LIN {X 0,Y 360.428,Z 320.263,A -85,B 0,C 180,E1 -13052.235,E2 -13052.235} C_VEL
LIN {X 0,Y 360.36,Z 319.532,A -85,B 0,C 180,E1 -13053.354,E2 -13053.354} C_VEL
LIN {X 0,Y 360.368,Z 318.39,A -85,B 0,C 180,E1 -13054.474,E2 -13054.474} C_VEL
LIN {X 0,Y 360.408,Z 314.81,A -85,B 0,C 180,E1 -13056.719,E2 -13056.719} C_VEL
LIN {X 0,Y 360.696,Z 310.966,A -85,B 0,C 180,E1 -13058.403,E2 -13058.403} C_VEL
LIN {X 0,Y 361.141,Z 306.012,A -85,B 0,C 180,E1 -13060.087,E2 -13060.087} C_VEL
LIN {X 0,Y 361.815,Z 299.808,A -85,B 0,C 180,E1 -13061.768,E2 -13061.768} C_VEL
LIN {X 0,Y 362.921,Z 292.123,A -85,B 0,C 180,E1 -13063.437,E2 -13063.437} C_VEL
LIN {X 0,Y 363.918,Z 283.845,A -85,B 0,C 180,E1 -13064.897,E2 -13064.897} C_VEL
LIN {X 0,Y 365.211,Z 273.678,A -85,B 0,C 180,E1 -13066.346,E2 -13066.346} C_VEL
LIN {X 0,Y 366.644,Z 262.906,A -85,B 0,C 180,E1 -13067.572,E2 -13067.572} C_VEL
LIN {X 0,Y 367.851,Z 252.444,A -85,B 0,C 180,E1 -13068.52,E2 -13068.52} C_VEL
LIN {X 0,Y 369.117,Z 239.88,A -85,B 0,C 180,E1 -13069.391,E2 -13069.391} C_VEL
LIN {X 0,Y 370.219,Z 226.622,A -85,B 0,C 180,E1 -13070.053,E2 -13070.053} C_VEL
LIN {X 0,Y 370.793,Z 214.493,A -85,B 0,C 180,E1 -13070.455,E2 -13070.455} C_VEL
LIN {X 0,Y 372.141,Z 144.791,A -85,B 0,C 180,E1 -13071.833,E2 -13071.833} C_VEL
LIN {X 0,Y 368.386,Z 121.336,A -85,B 0,C 180,E1 -13072.599,E2 -13072.599} C_VEL
LIN {X 0,Y 365.441,Z 106.485,A -85,B 0,C 180,E1 -13073.16,E2 -13073.16} C_VEL
LIN {X 0,Y 367.084,Z 91.512,A -85,B 0,C 180,E1 -13076.432,E2 -13076.432} C_VEL
LIN {X 0,Y 365.836,Z 84.095,A -85,B 0,C 180,E1 -13078.246,E2 -13078.246} C_VEL
LIN {X 0,Y 363.068,Z 72.33,A -85,B 0,C 180,E1 -13081.298,E2 -13081.298} C_VEL
LIN {X 0,Y 361.872,Z 67.409,A -85,B 0,C 180,E1 -13082.653,E2 -13082.653} C_VEL
LIN {X 0,Y 361.87,Z 67.409,A -85,B 0,C 180,E1 -13085.637,E2 -13085.637} C_VEL
LIN {X 0,Y 361.871,Z 67.398,A -85,B 0,C 180,E1 -13089.027,E2 -13089.027} C_VEL
LIN {X 0,Y 361.839,Z 67.408,A -85,B 0,C 180,E1 -13092.829,E2 -13092.829} C_VEL
LIN {X 0,Y 361.821,Z 67.412,A -85,B 0,C 180,E1 -13095.946,E2 -13095.946} C_VEL
LIN {X 0,Y 361.838,Z 67.41,A -85,B 0,C 180,E1 -13099.245,E2 -13099.245} C_VEL
LIN {X 0,Y 361.866,Z 67.404,A -85,B 0,C 180,E1 -13102.777,E2 -13102.777} C_VEL
LIN {X 0,Y 361.857,Z 67.405,A -85,B 0,C 180,E1 -13105.72,E2 -13105.72} C_VEL
LIN {X 0,Y 361.878,Z 67.401,A -85,B 0,C 180,E1 -13109.672,E2 -13109.672} C_VEL
LIN {X 0,Y 361.958,Z 67.392,A -85,B 0,C 180,E1 -13113.475,E2 -13113.475} C_VEL
LIN {X 0,Y 361.894,Z 67.402,A -85,B 0,C 180,E1 -13117.145,E2 -13117.145} C_VEL
LIN {X 0,Y 361.91,Z 67.405,A -85,B 0,C 180,E1 -13120.723,E2 -13120.723} C_VEL
LIN {X 0,Y 361.936,Z 67.392,A -85,B 0,C 180,E1 -13123.066,E2 -13123.066} C_VEL
LIN {X 0,Y 362.002,Z 67.389,A -85,B 0,C 180,E1 -13126.528,E2 -13126.528} C_VEL
LIN {X 0,Y 362.035,Z 67.387,A -85,B 0,C 180,E1 -13129.938,E2 -13129.938} C_VEL
LIN {X 0,Y 362.165,Z 67.36,A -85,B 0,C 180,E1 -13133.314,E2 -13133.314} C_VEL
LIN {X 0,Y 362.282,Z 67.351,A -85,B 0,C 180,E1 -13137.776,E2 -13137.776} C_VEL
LIN {X 0,Y 362.43,Z 67.338,A -85,B 0,C 180,E1 -13140,E2 -13140} C_VEL
LIN {X 0,Y 362.283,Z 67.353,A -85,B 0,C 180,E1 -13142.223,E2 -13142.223} C_VEL
LIN {X 0,Y 362.15,Z 67.372,A -85,B 0,C 180,E1 -13146.686,E2 -13146.686} C_VEL
LIN {X 0,Y 362.003,Z 67.389,A -85,B 0,C 180,E1 -13150.063,E2 -13150.063} C_VEL
LIN {X 0,Y 362.001,Z 67.383,A -85,B 0,C 180,E1 -13153.899,E2 -13153.899} C_VEL
LIN {X 0,Y 361.931,Z 67.404,A -85,B 0,C 180,E1 -13156.934,E2 -13156.934} C_VEL
LIN {X 0,Y 361.896,Z 67.404,A -85,B 0,C 180,E1 -13160.46,E2 -13160.46} C_VEL
LIN {X 0,Y 361.895,Z 67.401,A -85,B 0,C 180,E1 -13164.113,E2 -13164.113} C_VEL
LIN {X 0,Y 361.867,Z 67.405,A -85,B 0,C 180,E1 -13167.782,E2 -13167.782} C_VEL
LIN {X 0,Y 361.848,Z 67.409,A -85,B 0,C 180,E1 -13171.285,E2 -13171.285} C_VEL
LIN {X 0,Y 361.856,Z 67.408,A -85,B 0,C 180,E1 -13174.28,E2 -13174.28} C_VEL
LIN {X 0,Y 361.862,Z 67.407,A -85,B 0,C 180,E1 -13177.222,E2 -13177.222} C_VEL
LIN {X 0,Y 361.83,Z 67.4,A -85,B 0,C 180,E1 -13180.754,E2 -13180.754} C_VEL
LIN {X 0,Y 361.818,Z 67.416,A -85,B 0,C 180,E1 -13184.368,E2 -13184.368} C_VEL
LIN {X 0,Y 361.836,Z 67.416,A -85,B 0,C 180,E1 -13187.568,E2 -13187.568} C_VEL
LIN {X 0,Y 361.831,Z 67.413,A -85,B 0,C 180,E1 -13190.981,E2 -13190.981} C_VEL
LIN {X 0,Y 361.875,Z 67.411,A -85,B 0,C 180,E1 -13194.655,E2 -13194.655} C_VEL
LIN {X 0,Y 361.926,Z 67.537,A -85,B 0,C 180,E1 -13195.305,E2 -13195.305} C_VEL
LIN {X 0,Y 362.975,Z 72.103,A -85,B 0,C 180,E1 -13196.708,E2 -13196.708} C_VEL
LIN {X 0,Y 372.386,Z 94.109,A -85,B 0,C 180,E1 -13197.911,E2 -13197.911} C_VEL
LIN {X 0,Y 373.147,Z 96.414,A -85,B 0,C 180,E1 -13198.016,E2 -13198.016} C_VEL
LIN {X 0,Y 371.369,Z 178.271,A -85,B 0,C 180,E1 -13199.626,E2 -13199.626} C_VEL
LIN {X 0,Y 370.873,Z 191.183,A -85,B 0,C 180,E1 -13200.091,E2 -13200.091} C_VEL
LIN {X 0,Y 370.25,Z 203.565,A -85,B 0,C 180,E1 -13200.76,E2 -13200.76} C_VEL
LIN {X 0,Y 369.334,Z 215.148,A -85,B 0,C 180,E1 -13201.594,E2 -13201.594} C_VEL
LIN {X 0,Y 368.036,Z 227.162,A -85,B 0,C 180,E1 -13202.722,E2 -13202.722} C_VEL
LIN {X 0,Y 366.749,Z 238.059,A -85,B 0,C 180,E1 -13204.027,E2 -13204.027} C_VEL
LIN {X 0,Y 365.655,Z 246.559,A -85,B 0,C 180,E1 -13205.289,E2 -13205.289} C_VEL
LIN {X 0,Y 364.569,Z 254.494,A -85,B 0,C 180,E1 -13206.722,E2 -13206.722} C_VEL
LIN {X 0,Y 363.432,Z 262.175,A -85,B 0,C 180,E1 -13208.443,E2 -13208.443} C_VEL
LIN {X 0,Y 362.508,Z 268.298,A -85,B 0,C 180,E1 -13210.167,E2 -13210.167} C_VEL
LIN {X 0,Y 361.747,Z 273.775,A -85,B 0,C 180,E1 -13212.17,E2 -13212.17} C_VEL
LIN {X 0,Y 361.11,Z 277.706,A -85,B 0,C 180,E1 -13214.189,E2 -13214.189} C_VEL
LIN {X 0,Y 360.871,Z 279.318,A -85,B 0,C 180,E1 -13215.334,E2 -13215.334} C_VEL
LIN {X 0,Y 360.663,Z 280.878,A -85,B 0,C 180,E1 -13216.986,E2 -13216.986} C_VEL
LIN {X 0,Y 360.463,Z 281.603,A -85,B 0,C 180,E1 -13218.757,E2 -13218.757} C_VEL
LIN {X 0,Y 360.418,Z 281.121,A -85,B 0,C 180,E1 -13221.025,E2 -13221.025} C_VEL
LIN {X 0,Y 360.479,Z 280.243,A -85,B 0,C 180,E1 -13222.156,E2 -13222.156} C_VEL
LIN {X 0,Y 360.701,Z 278.598,A -85,B 0,C 180,E1 -13223.564,E2 -13223.564} C_VEL
LIN {X 0,Y 360.784,Z 275.189,A -85,B 0,C 180,E1 -13225.531,E2 -13225.531} C_VEL
LIN {X 0,Y 361.162,Z 271.131,A -85,B 0,C 180,E1 -13227.212,E2 -13227.212} C_VEL
LIN {X 0,Y 361.536,Z 264.937,A -85,B 0,C 180,E1 -13229.165,E2 -13229.165} C_VEL
LIN {X 0,Y 362.237,Z 258.176,A -85,B 0,C 180,E1 -13230.834,E2 -13230.834} C_VEL
LIN {X 0,Y 362.96,Z 249.785,A -85,B 0,C 180,E1 -13232.497,E2 -13232.497} C_VEL
LIN {X 0,Y 363.635,Z 241.169,A -85,B 0,C 180,E1 -13233.879,E2 -13233.879} C_VEL
LIN {X 0,Y 364.669,Z 231.668,A -85,B 0,C 180,E1 -13235.114,E2 -13235.114} C_VEL
LIN {X 0,Y 365.605,Z 219.921,A -85,B 0,C 180,E1 -13236.346,E2 -13236.346} C_VEL
LIN {X 0,Y 366.344,Z 208.102,A -85,B 0,C 180,E1 -13237.302,E2 -13237.302} C_VEL
LIN {X 0,Y 366.964,Z 195.817,A -85,B 0,C 180,E1 -13238.051,E2 -13238.051} C_VEL
LIN {X 0,Y 367.419,Z 183.163,A -85,B 0,C 180,E1 -13238.595,E2 -13238.595} C_VEL
LIN {X 0,Y 367.681,Z 169.87,A -85,B 0,C 180,E1 -13238.935,E2 -13238.935} C_VEL
LIN {X 0,Y 368.729,Z 92.38,A -85,B 0,C 180,E1 -13240.44,E2 -13240.44} C_VEL
LIN {X 0,Y 367.749,Z 87.16,A -85,B 0,C 180,E1 -13240.594,E2 -13240.594} C_VEL
LIN {X 0,Y 366.313,Z 83.319,A -85,B 0,C 180,E1 -13240.763,E2 -13240.763} C_VEL
LIN {X 0,Y 363.096,Z 78.907,A -85,B 0,C 180,E1 -13241.018,E2 -13241.018} C_VEL
LIN {X 0,Y 355.906,Z 71.842,A -85,B 0,C 180,E1 -13241.552,E2 -13241.552} C_VEL
LIN {X 0,Y 355.497,Z 71.151,A -85,B 0,C 180,E1 -13241.683,E2 -13241.683} C_VEL
LIN {X 0,Y 354.913,Z 68.277,A -85,B 0,C 180,E1 -13242.509,E2 -13242.509} C_VEL
LIN {X 0,Y 354.921,Z 68.274,A -85,B 0,C 180,E1 -13244.917,E2 -13244.917} C_VEL
LIN {X 0,Y 354.908,Z 68.279,A -85,B 0,C 180,E1 -13248.472,E2 -13248.472} C_VEL
LIN {X 0,Y 354.819,Z 68.288,A -85,B 0,C 180,E1 -13252.107,E2 -13252.107} C_VEL
LIN {X 0,Y 354.9,Z 68.277,A -85,B 0,C 180,E1 -13255.828,E2 -13255.828} C_VEL
LIN {X 0,Y 354.819,Z 68.287,A -85,B 0,C 180,E1 -13259.682,E2 -13259.682} C_VEL
LIN {X 0,Y 354.807,Z 68.29,A -85,B 0,C 180,E1 -13263.702,E2 -13263.702} C_VEL
LIN {X 0,Y 354.803,Z 68.287,A -85,B 0,C 180,E1 -13266.459,E2 -13266.459} C_VEL
LIN {X 0,Y 354.826,Z 68.287,A -85,B 0,C 180,E1 -13269.424,E2 -13269.424} C_VEL
LIN {X 0,Y 354.79,Z 68.288,A -85,B 0,C 180,E1 -13272.868,E2 -13272.868} C_VEL
LIN {X 0,Y 354.769,Z 68.291,A -85,B 0,C 180,E1 -13276.104,E2 -13276.104} C_VEL
LIN {X 0,Y 354.79,Z 68.292,A -85,B 0,C 180,E1 -13279.179,E2 -13279.179} C_VEL
LIN {X 0,Y 354.81,Z 68.285,A -85,B 0,C 180,E1 -13282.403,E2 -13282.403} C_VEL
LIN {X 0,Y 354.815,Z 68.289,A -85,B 0,C 180,E1 -13284.941,E2 -13284.941} C_VEL
LIN {X 0,Y 354.796,Z 68.288,A -85,B 0,C 180,E1 -13288.405,E2 -13288.405} C_VEL
LIN {X 0,Y 354.85,Z 68.281,A -85,B 0,C 180,E1 -13291.619,E2 -13291.619} C_VEL
LIN {X 0,Y 354.903,Z 68.274,A -85,B 0,C 180,E1 -13294.173,E2 -13294.173} C_VEL
LIN {X 0,Y 354.84,Z 68.282,A -85,B 0,C 180,E1 -13297.894,E2 -13297.894} C_VEL
LIN {X 0,Y 354.926,Z 68.272,A -85,B 0,C 180,E1 -13301.892,E2 -13301.892} C_VEL
LIN {X 0,Y 354.947,Z 68.27,A -85,B 0,C 180,E1 -13305.981,E2 -13305.981} C_VEL
LIN {X 0,Y 354.961,Z 68.268,A -85,B 0,C 180,E1 -13309.736,E2 -13309.736} C_VEL
LIN {X 0,Y 355.125,Z 68.246,A -85,B 0,C 180,E1 -13313.181,E2 -13313.181} C_VEL
LIN {X 0,Y 355.246,Z 68.235,A -85,B 0,C 180,E1 -13317.733,E2 -13317.733} C_VEL
LIN {X 0,Y 355.401,Z 68.216,A -85,B 0,C 180,E1 -13320,E2 -13320} C_VEL
LIN {X 0,Y 355.248,Z 68.232,A -85,B 0,C 180,E1 -13322.268,E2 -13322.268} C_VEL
LIN {X 0,Y 355.094,Z 68.25,A -85,B 0,C 180,E1 -13326.82,E2 -13326.82} C_VEL
LIN {X 0,Y 354.961,Z 68.267,A -85,B 0,C 180,E1 -13330.265,E2 -13330.265} C_VEL
LIN {X 0,Y 354.947,Z 68.269,A -85,B 0,C 180,E1 -13334.019,E2 -13334.019} C_VEL
LIN {X 0,Y 354.894,Z 68.275,A -85,B 0,C 180,E1 -13338.092,E2 -13338.092} C_VEL
LIN {X 0,Y 354.834,Z 68.282,A -85,B 0,C 180,E1 -13342.106,E2 -13342.106} C_VEL
LIN {X 0,Y 354.868,Z 68.278,A -85,B 0,C 180,E1 -13345.83,E2 -13345.83} C_VEL
LIN {X 0,Y 354.811,Z 68.285,A -85,B 0,C 180,E1 -13349.683,E2 -13349.683} C_VEL
LIN {X 0,Y 354.818,Z 68.284,A -85,B 0,C 180,E1 -13353.684,E2 -13353.684} C_VEL
LIN {X 0,Y 354.802,Z 68.291,A -85,B 0,C 180,E1 -13356.459,E2 -13356.459} C_VEL
LIN {X 0,Y 354.827,Z 68.283,A -85,B 0,C 180,E1 -13359.423,E2 -13359.423} C_VEL
LIN {X 0,Y 354.791,Z 68.289,A -85,B 0,C 180,E1 -13362.867,E2 -13362.867} C_VEL
LIN {X 0,Y 354.77,Z 68.295,A -85,B 0,C 180,E1 -13366.104,E2 -13366.104} C_VEL
LIN {X 0,Y 354.785,Z 68.288,A -85,B 0,C 180,E1 -13369.178,E2 -13369.178} C_VEL
LIN {X 0,Y 354.804,Z 68.288,A -85,B 0,C 180,E1 -13372.404,E2 -13372.404} C_VEL
LIN {X 0,Y 354.814,Z 68.285,A -85,B 0,C 180,E1 -13374.941,E2 -13374.941} C_VEL
LIN {X 0,Y 354.796,Z 68.288,A -85,B 0,C 180,E1 -13378.405,E2 -13378.405} C_VEL
LIN {X 0,Y 354.898,Z 68.48,A -85,B 0,C 180,E1 -13379.834,E2 -13379.834} C_VEL
LIN {X 0,Y 357.776,Z 82.272,A -85,B 0,C 180,E1 -13383.14,E2 -13383.14} C_VEL
LIN {X 0,Y 358.296,Z 86.562,A -85,B 0,C 180,E1 -13384.123,E2 -13384.123} C_VEL
LIN {X 0,Y 356.977,Z 101.67,A -85,B 0,C 180,E1 -13387.381,E2 -13387.381} C_VEL
LIN {X 0,Y 356.58,Z 106.923,A -85,B 0,C 180,E1 -13388.502,E2 -13388.502} C_VEL
LIN {X 0,Y 361.35,Z 145.103,A -85,B 0,C 180,E1 -13389.527,E2 -13389.527} C_VEL
LIN {X 0,Y 360.307,Z 216.41,A -85,B 0,C 180,E1 -13390.967,E2 -13390.967} C_VEL
LIN {X 0,Y 359.677,Z 230.303,A -85,B 0,C 180,E1 -13391.487,E2 -13391.487} C_VEL
LIN {X 0,Y 358.817,Z 242.738,A -85,B 0,C 180,E1 -13392.179,E2 -13392.179} C_VEL
LIN {X 0,Y 357.745,Z 255.455,A -85,B 0,C 180,E1 -13393.156,E2 -13393.156} C_VEL
LIN {X 0,Y 356.788,Z 266.794,A -85,B 0,C 180,E1 -13394.285,E2 -13394.285} C_VEL
LIN {X 0,Y 355.791,Z 277.222,A -85,B 0,C 180,E1 -13395.595,E2 -13395.595} C_VEL
LIN {X 0,Y 355.113,Z 285.356,A -85,B 0,C 180,E1 -13396.844,E2 -13396.844} C_VEL
LIN {X 0,Y 354.492,Z 293.09,A -85,B 0,C 180,E1 -13398.275,E2 -13398.275} C_VEL
LIN {X 0,Y 353.879,Z 300.655,A -85,B 0,C 180,E1 -13399.992,E2 -13399.992} C_VEL
LIN {X 0,Y 353.51,Z 307.638,A -85,B 0,C 180,E1 -13402,E2 -13402} C_VEL
LIN {X 0,Y 353.297,Z 312.985,A -85,B 0,C 180,E1 -13404.063,E2 -13404.063} C_VEL
LIN {X 0,Y 353.376,Z 315.715,A -85,B 0,C 180,E1 -13405.437,E2 -13405.437} C_VEL
LIN {X 0,Y 353.416,Z 318.756,A -85,B 0,C 180,E1 -13407.721,E2 -13407.721} C_VEL
LIN {X 0,Y 353.475,Z 319.67,A -85,B 0,C 180,E1 -13408.861,E2 -13408.861} C_VEL
LIN {X 0,Y 353.456,Z 320.167,A -85,B 0,C 180,E1 -13410,E2 -13410} C_VEL
LIN {X 0,Y 353.433,Z 320.231,A -85,B 0,C 180,E1 -13411.139,E2 -13411.139} C_VEL
LIN {X 0,Y 353.276,Z 319.19,A -85,B 0,C 180,E1 -13413.421,E2 -13413.421} C_VEL
LIN {X 0,Y 353.276,Z 318.08,A -85,B 0,C 180,E1 -13414.564,E2 -13414.564} C_VEL
LIN {X 0,Y 353.271,Z 316.217,A -85,B 0,C 180,E1 -13415.897,E2 -13415.897} C_VEL
LIN {X 0,Y 353.53,Z 312.141,A -85,B 0,C 180,E1 -13417.999,E2 -13417.999} C_VEL
LIN {X 0,Y 353.926,Z 307.614,A -85,B 0,C 180,E1 -13419.717,E2 -13419.717} C_VEL
LIN {X 0,Y 354.688,Z 300.798,A -85,B 0,C 180,E1 -13421.718,E2 -13421.718} C_VEL
LIN {X 0,Y 355.815,Z 293.418,A -85,B 0,C 180,E1 -13423.42,E2 -13423.42} C_VEL
LIN {X 0,Y 356.968,Z 284.469,A -85,B 0,C 180,E1 -13425.091,E2 -13425.091} C_VEL
LIN {X 0,Y 358.239,Z 274.846,A -85,B 0,C 180,E1 -13426.527,E2 -13426.527} C_VEL
LIN {X 0,Y 359.698,Z 264.397,A -85,B 0,C 180,E1 -13427.776,E2 -13427.776} C_VEL
LIN {X 0,Y 361.154,Z 252.806,A -85,B 0,C 180,E1 -13428.876,E2 -13428.876} C_VEL
LIN {X 0,Y 362.449,Z 240.521,A -85,B 0,C 180,E1 -13429.762,E2 -13429.762} C_VEL
LIN {X 0,Y 363.653,Z 226.863,A -85,B 0,C 180,E1 -13430.468,E2 -13430.468} C_VEL
LIN {X 0,Y 364.311,Z 213.85,A -85,B 0,C 180,E1 -13430.909,E2 -13430.909} C_VEL
LIN {X 0,Y 365.68,Z 145.475,A -85,B 0,C 180,E1 -13432.285,E2 -13432.285} C_VEL
LIN {X 0,Y 361.753,Z 121.278,A -85,B 0,C 180,E1 -13433.105,E2 -13433.105} C_VEL
LIN {X 0,Y 358.726,Z 106.105,A -85,B 0,C 180,E1 -13433.691,E2 -13433.691} C_VEL
LIN {X 0,Y 360.216,Z 92.799,A -85,B 0,C 180,E1 -13436.663,E2 -13436.663} C_VEL
LIN {X 0,Y 358.751,Z 84.671,A -85,B 0,C 180,E1 -13438.707,E2 -13438.707} C_VEL
LIN {X 0,Y 355.924,Z 72.749,A -85,B 0,C 180,E1 -13441.889,E2 -13441.889} C_VEL
LIN {X 0,Y 354.82,Z 68.289,A -85,B 0,C 180,E1 -13443.174,E2 -13443.174} C_VEL
LIN {X 0,Y 354.8,Z 68.289,A -85,B 0,C 180,E1 -13446.459,E2 -13446.459} C_VEL
LIN {X 0,Y 354.826,Z 68.274,A -85,B 0,C 180,E1 -13449.424,E2 -13449.424} C_VEL
LIN {X 0,Y 354.791,Z 68.286,A -85,B 0,C 180,E1 -13452.867,E2 -13452.867} C_VEL
LIN {X 0,Y 354.77,Z 68.289,A -85,B 0,C 180,E1 -13456.104,E2 -13456.104} C_VEL
LIN {X 0,Y 354.79,Z 68.288,A -85,B 0,C 180,E1 -13459.179,E2 -13459.179} C_VEL
LIN {X 0,Y 354.809,Z 68.282,A -85,B 0,C 180,E1 -13462.403,E2 -13462.403} C_VEL
LIN {X 0,Y 354.815,Z 68.286,A -85,B 0,C 180,E1 -13464.941,E2 -13464.941} C_VEL
LIN {X 0,Y 354.796,Z 68.289,A -85,B 0,C 180,E1 -13468.405,E2 -13468.405} C_VEL
LIN {X 0,Y 354.854,Z 68.282,A -85,B 0,C 180,E1 -13471.619,E2 -13471.619} C_VEL
LIN {X 0,Y 354.903,Z 68.269,A -85,B 0,C 180,E1 -13474.173,E2 -13474.173} C_VEL
LIN {X 0,Y 354.838,Z 68.279,A -85,B 0,C 180,E1 -13477.894,E2 -13477.894} C_VEL
LIN {X 0,Y 354.926,Z 68.271,A -85,B 0,C 180,E1 -13481.892,E2 -13481.892} C_VEL
LIN {X 0,Y 354.946,Z 68.272,A -85,B 0,C 180,E1 -13485.981,E2 -13485.981} C_VEL
LIN {X 0,Y 354.982,Z 68.264,A -85,B 0,C 180,E1 -13489.736,E2 -13489.736} C_VEL
LIN {X 0,Y 355.128,Z 68.236,A -85,B 0,C 180,E1 -13493.18,E2 -13493.18} C_VEL
LIN {X 0,Y 355.245,Z 68.227,A -85,B 0,C 180,E1 -13497.732,E2 -13497.732} C_VEL
LIN {X 0,Y 355.4,Z 68.214,A -85,B 0,C 180,E1 -13500,E2 -13500} C_VEL
LIN {X 0,Y 355.246,Z 68.229,A -85,B 0,C 180,E1 -13502.267,E2 -13502.267} C_VEL
LIN {X 0,Y 355.114,Z 68.249,A -85,B 0,C 180,E1 -13506.82,E2 -13506.82} C_VEL
LIN {X 0,Y 354.959,Z 68.266,A -85,B 0,C 180,E1 -13510.265,E2 -13510.265} C_VEL
LIN {X 0,Y 354.946,Z 68.262,A -85,B 0,C 180,E1 -13514.019,E2 -13514.019} C_VEL
LIN {X 0,Y 354.892,Z 68.271,A -85,B 0,C 180,E1 -13518.092,E2 -13518.092} C_VEL
LIN {X 0,Y 354.837,Z 68.282,A -85,B 0,C 180,E1 -13522.106,E2 -13522.106} C_VEL
LIN {X 0,Y 354.868,Z 68.279,A -85,B 0,C 180,E1 -13525.83,E2 -13525.83} C_VEL
LIN {X 0,Y 354.809,Z 68.286,A -85,B 0,C 180,E1 -13529.683,E2 -13529.683} C_VEL
LIN {X 0,Y 354.816,Z 68.284,A -85,B 0,C 180,E1 -13533.684,E2 -13533.684} C_VEL
LIN {X 0,Y 354.798,Z 68.288,A -85,B 0,C 180,E1 -13536.459,E2 -13536.459} C_VEL
LIN {X 0,Y 354.8,Z 68.288,A -85,B 0,C 180,E1 -13539.418,E2 -13539.418} C_VEL
LIN {X 0,Y 354.787,Z 68.293,A -85,B 0,C 180,E1 -13542.867,E2 -13542.867} C_VEL
LIN {X 0,Y 354.768,Z 68.295,A -85,B 0,C 180,E1 -13546.103,E2 -13546.103} C_VEL
LIN {X 0,Y 354.786,Z 68.293,A -85,B 0,C 180,E1 -13549.179,E2 -13549.179} C_VEL
LIN {X 0,Y 354.801,Z 68.291,A -85,B 0,C 180,E1 -13552.404,E2 -13552.404} C_VEL
LIN {X 0,Y 354.86,Z 68.405,A -85,B 0,C 180,E1 -13554.826,E2 -13554.826} C_VEL
LIN {X 0,Y 355.909,Z 72.666,A -85,B 0,C 180,E1 -13556.136,E2 -13556.136} C_VEL
LIN {X 0,Y 364.732,Z 92.87,A -85,B 0,C 180,E1 -13557.299,E2 -13557.299} C_VEL
LIN {X 0,Y 366.692,Z 97.801,A -85,B 0,C 180,E1 -13557.558,E2 -13557.558} C_VEL
LIN {X 0,Y 364.89,Z 178.971,A -85,B 0,C 180,E1 -13559.189,E2 -13559.189} C_VEL
LIN {X 0,Y 364.324,Z 192.551,A -85,B 0,C 180,E1 -13559.697,E2 -13559.697} C_VEL
LIN {X 0,Y 363.607,Z 205.559,A -85,B 0,C 180,E1 -13560.434,E2 -13560.434} C_VEL
LIN {X 0,Y 362.572,Z 217.275,A -85,B 0,C 180,E1 -13561.331,E2 -13561.331} C_VEL
LIN {X 0,Y 361.233,Z 228.942,A -85,B 0,C 180,E1 -13562.479,E2 -13562.479} C_VEL
LIN {X 0,Y 359.947,Z 239.253,A -85,B 0,C 180,E1 -13563.765,E2 -13563.765} C_VEL
LIN {X 0,Y 358.771,Z 247.845,A -85,B 0,C 180,E1 -13565.092,E2 -13565.092} C_VEL
LIN {X 0,Y 357.436,Z 256.987,A -85,B 0,C 180,E1 -13566.843,E2 -13566.843} C_VEL
LIN {X 0,Y 356.305,Z 264.287,A -85,B 0,C 180,E1 -13568.598,E2 -13568.598} C_VEL
LIN {X 0,Y 355.355,Z 270.039,A -85,B 0,C 180,E1 -13570.353,E2 -13570.353} C_VEL
LIN {X 0,Y 354.739,Z 274.241,A -85,B 0,C 180,E1 -13571.983,E2 -13571.983} C_VEL
LIN {X 0,Y 354.119,Z 277.882,A -85,B 0,C 180,E1 -13573.868,E2 -13573.868} C_VEL
LIN {X 0,Y 353.853,Z 279.534,A -85,B 0,C 180,E1 -13575.037,E2 -13575.037} C_VEL
LIN {X 0,Y 353.592,Z 281.284,A -85,B 0,C 180,E1 -13576.887,E2 -13576.887} C_VEL
LIN {X 0,Y 353.41,Z 281.972,A -85,B 0,C 180,E1 -13578.53,E2 -13578.53} C_VEL
LIN {X 0,Y 353.329,Z 281.57,A -85,B 0,C 180,E1 -13580.844,E2 -13580.844} C_VEL
LIN {X 0,Y 353.394,Z 280.762,A -85,B 0,C 180,E1 -13581.998,E2 -13581.998} C_VEL
LIN {X 0,Y 353.62,Z 278.974,A -85,B 0,C 180,E1 -13583.577,E2 -13583.577} C_VEL
LIN {X 0,Y 353.701,Z 275.85,A -85,B 0,C 180,E1 -13585.441,E2 -13585.441} C_VEL
LIN {X 0,Y 354.064,Z 271.878,A -85,B 0,C 180,E1 -13587.156,E2 -13587.156} C_VEL
LIN {X 0,Y 354.457,Z 265.792,A -85,B 0,C 180,E1 -13589.148,E2 -13589.148} C_VEL
LIN {X 0,Y 355.18,Z 259.133,A -85,B 0,C 180,E1 -13590.85,E2 -13590.85} C_VEL
LIN {X 0,Y 355.893,Z 250.908,A -85,B 0,C 180,E1 -13592.547,E2 -13592.547} C_VEL
LIN {X 0,Y 356.593,Z 242.464,A -85,B 0,C 180,E1 -13593.956,E2 -13593.956} C_VEL
LIN {X 0,Y 357.754,Z 231.982,A -85,B 0,C 180,E1 -13595.354,E2 -13595.354} C_VEL
LIN {X 0,Y 358.622,Z 221.64,A -85,B 0,C 180,E1 -13596.47,E2 -13596.47} C_VEL
LIN {X 0,Y 359.408,Z 210.303,A -85,B 0,C 180,E1 -13597.444,E2 -13597.444} C_VEL
LIN {X 0,Y 360.007,Z 198.626,A -85,B 0,C 180,E1 -13598.207,E2 -13598.207} C_VEL
LIN {X 0,Y 360.517,Z 185.179,A -85,B 0,C 180,E1 -13598.831,E2 -13598.831} C_VEL
LIN {X 0,Y 360.852,Z 173.211,A -85,B 0,C 180,E1 -13599.176,E2 -13599.176} C_VEL
LIN {X 0,Y 361.944,Z 93.039,A -85,B 0,C 180,E1 -13600.766,E2 -13600.766} C_VEL
LIN {X 0,Y 360.102,Z 85.21,A -85,B 0,C 180,E1 -13601.022,E2 -13601.022} C_VEL
LIN {X 0,Y 355.571,Z 71.513,A -85,B 0,C 180,E1 -13601.58,E2 -13601.58} C_VEL
LIN {X 0,Y 355.497,Z 71.151,A -85,B 0,C 180,E1 -13601.683,E2 -13601.683} C_VEL
LIN {X 0,Y 354.86,Z 69.684,A -85,B 0,C 180,E1 -13602.249,E2 -13602.249} C_VEL
LIN {X 0,Y 353.838,Z 68.938,A -85,B 0,C 180,E1 -13602.842,E2 -13602.842} C_VEL
LIN {X 0,Y 351.292,Z 68.726,A -85,B 0,C 180,E1 -13604.059,E2 -13604.059} C_VEL
LIN {X 0,Y 348.907,Z 69.021,A -85,B 0,C 180,E1 -13605.335,E2 -13605.335} C_VEL
LIN {X 0,Y 347.916,Z 69.15,A -85,B 0,C 180,E1 -13606.323,E2 -13606.323} C_VEL
LIN {X 0,Y 347.834,Z 69.157,A -85,B 0,C 180,E1 -13606.656,E2 -13606.656} C_VEL
LIN {X 0,Y 347.857,Z 69.153,A -85,B 0,C 180,E1 -13608.86,E2 -13608.86} C_VEL
LIN {X 0,Y 347.765,Z 69.166,A -85,B 0,C 180,E1 -13612.58,E2 -13612.58} C_VEL
LIN {X 0,Y 347.812,Z 69.157,A -85,B 0,C 180,E1 -13615.109,E2 -13615.109} C_VEL
LIN {X 0,Y 347.811,Z 69.159,A -85,B 0,C 180,E1 -13617.694,E2 -13617.694} C_VEL
LIN {X 0,Y 347.75,Z 69.167,A -85,B 0,C 180,E1 -13620.348,E2 -13620.348} C_VEL
LIN {X 0,Y 347.75,Z 69.169,A -85,B 0,C 180,E1 -13624.044,E2 -13624.044} C_VEL
LIN {X 0,Y 347.768,Z 69.164,A -85,B 0,C 180,E1 -13627.32,E2 -13627.32} C_VEL
LIN {X 0,Y 347.735,Z 69.167,A -85,B 0,C 180,E1 -13630.297,E2 -13630.297} C_VEL
LIN {X 0,Y 347.725,Z 69.172,A -85,B 0,C 180,E1 -13633.408,E2 -13633.408} C_VEL
LIN {X 0,Y 347.727,Z 69.168,A -85,B 0,C 180,E1 -13636.687,E2 -13636.687} C_VEL
LIN {X 0,Y 347.749,Z 69.165,A -85,B 0,C 180,E1 -13640.173,E2 -13640.173} C_VEL
LIN {X 0,Y 347.764,Z 69.164,A -85,B 0,C 180,E1 -13642.68,E2 -13642.68} C_VEL
LIN {X 0,Y 347.751,Z 69.165,A -85,B 0,C 180,E1 -13645.957,E2 -13645.957} C_VEL
LIN {X 0,Y 347.752,Z 69.165,A -85,B 0,C 180,E1 -13649.652,E2 -13649.652} C_VEL
LIN {X 0,Y 347.834,Z 69.154,A -85,B 0,C 180,E1 -13653.608,E2 -13653.608} C_VEL
LIN {X 0,Y 347.793,Z 69.16,A -85,B 0,C 180,E1 -13656.162,E2 -13656.162} C_VEL
LIN {X 0,Y 347.817,Z 69.157,A -85,B 0,C 180,E1 -13659.91,E2 -13659.91} C_VEL
LIN {X 0,Y 347.87,Z 69.154,A -85,B 0,C 180,E1 -13662.36,E2 -13662.36} C_VEL
LIN {X 0,Y 347.901,Z 69.148,A -85,B 0,C 180,E1 -13665.971,E2 -13665.971} C_VEL
LIN {X 0,Y 347.901,Z 69.146,A -85,B 0,C 180,E1 -13669.525,E2 -13669.525} C_VEL
LIN {X 0,Y 348.092,Z 69.122,A -85,B 0,C 180,E1 -13673.042,E2 -13673.042} C_VEL
LIN {X 0,Y 348.208,Z 69.111,A -85,B 0,C 180,E1 -13677.687,E2 -13677.687} C_VEL
LIN {X 0,Y 348.349,Z 69.094,A -85,B 0,C 180,E1 -13680,E2 -13680} C_VEL
LIN {X 0,Y 348.21,Z 69.109,A -85,B 0,C 180,E1 -13682.314,E2 -13682.314} C_VEL
LIN {X 0,Y 348.061,Z 69.127,A -85,B 0,C 180,E1 -13686.959,E2 -13686.959} C_VEL
LIN {X 0,Y 347.901,Z 69.146,A -85,B 0,C 180,E1 -13690.475,E2 -13690.475} C_VEL
LIN {X 0,Y 347.903,Z 69.146,A -85,B 0,C 180,E1 -13694.15,E2 -13694.15} C_VEL
LIN {X 0,Y 347.833,Z 69.154,A -85,B 0,C 180,E1 -13698.259,E2 -13698.259} C_VEL
LIN {X 0,Y 347.79,Z 69.161,A -85,B 0,C 180,E1 -13701.634,E2 -13701.634} C_VEL
LIN {X 0,Y 347.797,Z 69.163,A -85,B 0,C 180,E1 -13705.11,E2 -13705.11} C_VEL
LIN {X 0,Y 347.761,Z 69.167,A -85,B 0,C 180,E1 -13709.014,E2 -13709.014} C_VEL
LIN {X 0,Y 347.737,Z 69.168,A -85,B 0,C 180,E1 -13713.072,E2 -13713.072} C_VEL
LIN {X 0,Y 347.774,Z 69.163,A -85,B 0,C 180,E1 -13716.065,E2 -13716.065} C_VEL
LIN {X 0,Y 347.755,Z 69.167,A -85,B 0,C 180,E1 -13718.793,E2 -13718.793} C_VEL
LIN {X 0,Y 347.754,Z 69.166,A -85,B 0,C 180,E1 -13721.83,E2 -13721.83} C_VEL
LIN {X 0,Y 347.709,Z 69.17,A -85,B 0,C 180,E1 -13725.027,E2 -13725.027} C_VEL
LIN {X 0,Y 347.75,Z 69.168,A -85,B 0,C 180,E1 -13728.398,E2 -13728.398} C_VEL
LIN {X 0,Y 347.767,Z 69.168,A -85,B 0,C 180,E1 -13732.013,E2 -13732.013} C_VEL
LIN {X 0,Y 347.747,Z 69.168,A -85,B 0,C 180,E1 -13735.536,E2 -13735.536} C_VEL
LIN {X 0,Y 347.843,Z 69.318,A -85,B 0,C 180,E1 -13739.535,E2 -13739.535} C_VEL
LIN {X 0,Y 350.423,Z 81.487,A -85,B 0,C 180,E1 -13742.53,E2 -13742.53} C_VEL
LIN {X 0,Y 351.322,Z 87.231,A -85,B 0,C 180,E1 -13743.89,E2 -13743.89} C_VEL
LIN {X 0,Y 350.094,Z 101.428,A -85,B 0,C 180,E1 -13747.017,E2 -13747.017} C_VEL
LIN {X 0,Y 349.661,Z 106.463,A -85,B 0,C 180,E1 -13748.119,E2 -13748.119} C_VEL
LIN {X 0,Y 354.574,Z 145.959,A -85,B 0,C 180,E1 -13749.214,E2 -13749.214} C_VEL
LIN {X 0,Y 353.491,Z 216.217,A -85,B 0,C 180,E1 -13750.661,E2 -13750.661} C_VEL
LIN {X 0,Y 352.814,Z 230.041,A -85,B 0,C 180,E1 -13751.188,E2 -13751.188} C_VEL
LIN {X 0,Y 351.94,Z 242.439,A -85,B 0,C 180,E1 -13751.894,E2 -13751.894} C_VEL
LIN {X 0,Y 350.963,Z 254.346,A -85,B 0,C 180,E1 -13752.82,E2 -13752.82} C_VEL
LIN {X 0,Y 349.884,Z 265.807,A -85,B 0,C 180,E1 -13753.967,E2 -13753.967} C_VEL
LIN {X 0,Y 348.902,Z 276.389,A -85,B 0,C 180,E1 -13755.304,E2 -13755.304} C_VEL
LIN {X 0,Y 348.168,Z 284.595,A -85,B 0,C 180,E1 -13756.577,E2 -13756.577} C_VEL
LIN {X 0,Y 347.362,Z 293.764,A -85,B 0,C 180,E1 -13758.327,E2 -13758.327} C_VEL
LIN {X 0,Y 346.756,Z 301.144,A -85,B 0,C 180,E1 -13760.08,E2 -13760.08} C_VEL
LIN {X 0,Y 346.46,Z 307.056,A -85,B 0,C 180,E1 -13761.836,E2 -13761.836} C_VEL
LIN {X 0,Y 346.201,Z 311.822,A -85,B 0,C 180,E1 -13763.648,E2 -13763.648} C_VEL
LIN {X 0,Y 346.28,Z 315.216,A -85,B 0,C 180,E1 -13765.343,E2 -13765.343} C_VEL
LIN {X 0,Y 346.251,Z 316.971,A -85,B 0,C 180,E1 -13766.509,E2 -13766.509} C_VEL
LIN {X 0,Y 346.318,Z 318.306,A -85,B 0,C 180,E1 -13767.674,E2 -13767.674} C_VEL
LIN {X 0,Y 346.411,Z 319.241,A -85,B 0,C 180,E1 -13768.837,E2 -13768.837} C_VEL
LIN {X 0,Y 346.393,Z 319.768,A -85,B 0,C 180,E1 -13770,E2 -13770} C_VEL
LIN {X 0,Y 346.351,Z 319.856,A -85,B 0,C 180,E1 -13771.163,E2 -13771.163} C_VEL
LIN {X 0,Y 346.194,Z 318.85,A -85,B 0,C 180,E1 -13773.492,E2 -13773.492} C_VEL
LIN {X 0,Y 346.189,Z 317.765,A -85,B 0,C 180,E1 -13774.658,E2 -13774.658} C_VEL
LIN {X 0,Y 346.198,Z 316.141,A -85,B 0,C 180,E1 -13775.885,E2 -13775.885} C_VEL
LIN {X 0,Y 346.482,Z 311.895,A -85,B 0,C 180,E1 -13778.163,E2 -13778.163} C_VEL
LIN {X 0,Y 346.89,Z 307.41,A -85,B 0,C 180,E1 -13779.916,E2 -13779.916} C_VEL
LIN {X 0,Y 347.71,Z 300.664,A -85,B 0,C 180,E1 -13781.957,E2 -13781.957} C_VEL
LIN {X 0,Y 348.888,Z 293.339,A -85,B 0,C 180,E1 -13783.691,E2 -13783.691} C_VEL
LIN {X 0,Y 350.016,Z 285.054,A -85,B 0,C 180,E1 -13785.288,E2 -13785.288} C_VEL
LIN {X 0,Y 351.301,Z 275.973,A -85,B 0,C 180,E1 -13786.713,E2 -13786.713} C_VEL
LIN {X 0,Y 352.783,Z 265.896,A -85,B 0,C 180,E1 -13787.986,E2 -13787.986} C_VEL
LIN {X 0,Y 354.247,Z 254.736,A -85,B 0,C 180,E1 -13789.108,E2 -13789.108} C_VEL
LIN {X 0,Y 355.68,Z 242.236,A -85,B 0,C 180,E1 -13790.079,E2 -13790.079} C_VEL
LIN {X 0,Y 356.91,Z 229.432,A -85,B 0,C 180,E1 -13790.797,E2 -13790.797} C_VEL
LIN {X 0,Y 357.707,Z 216.947,A -85,B 0,C 180,E1 -13791.276,E2 -13791.276} C_VEL
LIN {X 0,Y 358.363,Z 194.782,A -85,B 0,C 180,E1 -13791.764,E2 -13791.764} C_VEL
LIN {X 0,Y 359.305,Z 146.569,A -85,B 0,C 180,E1 -13792.743,E2 -13792.743} C_VEL
LIN {X 0,Y 355.547,Z 123.289,A -85,B 0,C 180,E1 -13793.552,E2 -13793.552} C_VEL
LIN {X 0,Y 352.012,Z 105.652,A -85,B 0,C 180,E1 -13794.263,E2 -13794.263} C_VEL
LIN {X 0,Y 353.312,Z 94.836,A -85,B 0,C 180,E1 -13796.724,E2 -13796.724} C_VEL
LIN {X 0,Y 352.371,Z 88.426,A -85,B 0,C 180,E1 -13798.35,E2 -13798.35} C_VEL
LIN {X 0,Y 349.655,Z 76.732,A -85,B 0,C 180,E1 -13801.507,E2 -13801.507} C_VEL
LIN {X 0,Y 347.775,Z 69.165,A -85,B 0,C 180,E1 -13803.679,E2 -13803.679} C_VEL
LIN {X 0,Y 347.764,Z 69.166,A -85,B 0,C 180,E1 -13807.321,E2 -13807.321} C_VEL
LIN {X 0,Y 347.735,Z 69.162,A -85,B 0,C 180,E1 -13810.297,E2 -13810.297} C_VEL
LIN {X 0,Y 347.725,Z 69.169,A -85,B 0,C 180,E1 -13813.408,E2 -13813.408} C_VEL
LIN {X 0,Y 347.728,Z 69.165,A -85,B 0,C 180,E1 -13816.686,E2 -13816.686} C_VEL
LIN {X 0,Y 347.75,Z 69.159,A -85,B 0,C 180,E1 -13820.173,E2 -13820.173} C_VEL
LIN {X 0,Y 347.764,Z 69.161,A -85,B 0,C 180,E1 -13822.679,E2 -13822.679} C_VEL
LIN {X 0,Y 347.751,Z 69.161,A -85,B 0,C 180,E1 -13825.956,E2 -13825.956} C_VEL
LIN {X 0,Y 347.767,Z 69.159,A -85,B 0,C 180,E1 -13829.654,E2 -13829.654} C_VEL
LIN {X 0,Y 347.855,Z 69.156,A -85,B 0,C 180,E1 -13832.745,E2 -13832.745} C_VEL
LIN {X 0,Y 347.792,Z 69.161,A -85,B 0,C 180,E1 -13836.162,E2 -13836.162} C_VEL
LIN {X 0,Y 347.816,Z 69.156,A -85,B 0,C 180,E1 -13839.909,E2 -13839.909} C_VEL
LIN {X 0,Y 347.87,Z 69.147,A -85,B 0,C 180,E1 -13842.359,E2 -13842.359} C_VEL
LIN {X 0,Y 347.901,Z 69.149,A -85,B 0,C 180,E1 -13845.971,E2 -13845.971} C_VEL
LIN {X 0,Y 347.932,Z 69.141,A -85,B 0,C 180,E1 -13849.526,E2 -13849.526} C_VEL
LIN {X 0,Y 348.094,Z 69.112,A -85,B 0,C 180,E1 -13853.042,E2 -13853.042} C_VEL
LIN {X 0,Y 348.207,Z 69.104,A -85,B 0,C 180,E1 -13857.686,E2 -13857.686} C_VEL
LIN {X 0,Y 348.348,Z 69.092,A -85,B 0,C 180,E1 -13860,E2 -13860} C_VEL
LIN {X 0,Y 348.209,Z 69.105,A -85,B 0,C 180,E1 -13862.313,E2 -13862.313} C_VEL
LIN {X 0,Y 348.08,Z 69.126,A -85,B 0,C 180,E1 -13866.958,E2 -13866.958} C_VEL
LIN {X 0,Y 347.9,Z 69.146,A -85,B 0,C 180,E1 -13870.475,E2 -13870.475} C_VEL
LIN {X 0,Y 347.901,Z 69.139,A -85,B 0,C 180,E1 -13874.15,E2 -13874.15} C_VEL
LIN {X 0,Y 347.832,Z 69.151,A -85,B 0,C 180,E1 -13878.259,E2 -13878.259} C_VEL
LIN {X 0,Y 347.791,Z 69.16,A -85,B 0,C 180,E1 -13881.635,E2 -13881.635} C_VEL
LIN {X 0,Y 347.797,Z 69.163,A -85,B 0,C 180,E1 -13885.11,E2 -13885.11} C_VEL
LIN {X 0,Y 347.759,Z 69.167,A -85,B 0,C 180,E1 -13889.014,E2 -13889.014} C_VEL
LIN {X 0,Y 347.734,Z 69.167,A -85,B 0,C 180,E1 -13893.072,E2 -13893.072} C_VEL
LIN {X 0,Y 347.771,Z 69.167,A -85,B 0,C 180,E1 -13896.065,E2 -13896.065} C_VEL
LIN {X 0,Y 347.732,Z 69.17,A -85,B 0,C 180,E1 -13898.795,E2 -13898.795} C_VEL
LIN {X 0,Y 347.748,Z 69.158,A -85,B 0,C 180,E1 -13901.831,E2 -13901.831} C_VEL
LIN {X 0,Y 347.707,Z 69.174,A -85,B 0,C 180,E1 -13905.027,E2 -13905.027} C_VEL
LIN {X 0,Y 347.75,Z 69.169,A -85,B 0,C 180,E1 -13908.397,E2 -13908.397} C_VEL
LIN {X 0,Y 347.764,Z 69.167,A -85,B 0,C 180,E1 -13912.013,E2 -13912.013} C_VEL
LIN {X 0,Y 347.801,Z 69.192,A -85,B 0,C 180,E1 -13914.305,E2 -13914.305} C_VEL
LIN {X 0,Y 348.712,Z 73.076,A -85,B 0,C 180,E1 -13915.521,E2 -13915.521} C_VEL
LIN {X 0,Y 357.165,Z 91.838,A -85,B 0,C 180,E1 -13916.669,E2 -13916.669} C_VEL
LIN {X 0,Y 360.265,Z 99.45,A -85,B 0,C 180,E1 -13917.088,E2 -13917.088} C_VEL
LIN {X 0,Y 358.43,Z 179.721,A -85,B 0,C 180,E1 -13918.735,E2 -13918.735} C_VEL
LIN {X 0,Y 357.841,Z 193.183,A -85,B 0,C 180,E1 -13919.252,E2 -13919.252} C_VEL
LIN {X 0,Y 357.107,Z 205.939,A -85,B 0,C 180,E1 -13919.99,E2 -13919.99} C_VEL
LIN {X 0,Y 356.018,Z 217.791,A -85,B 0,C 180,E1 -13920.915,E2 -13920.915} C_VEL
LIN {X 0,Y 354.608,Z 229.43,A -85,B 0,C 180,E1 -13922.081,E2 -13922.081} C_VEL
LIN {X 0,Y 353.337,Z 239.224,A -85,B 0,C 180,E1 -13923.32,E2 -13923.32} C_VEL
LIN {X 0,Y 352.141,Z 247.439,A -85,B 0,C 180,E1 -13924.59,E2 -13924.59} C_VEL
LIN {X 0,Y 350.959,Z 255.349,A -85,B 0,C 180,E1 -13926.077,E2 -13926.077} C_VEL
LIN {X 0,Y 349.678,Z 263.011,A -85,B 0,C 180,E1 -13927.861,E2 -13927.861} C_VEL
LIN {X 0,Y 348.5,Z 270.031,A -85,B 0,C 180,E1 -13929.951,E2 -13929.951} C_VEL
LIN {X 0,Y 347.748,Z 274.689,A -85,B 0,C 180,E1 -13931.782,E2 -13931.782} C_VEL
LIN {X 0,Y 347.151,Z 278.057,A -85,B 0,C 180,E1 -13933.535,E2 -13933.535} C_VEL
LIN {X 0,Y 346.845,Z 279.75,A -85,B 0,C 180,E1 -13934.727,E2 -13934.727} C_VEL
LIN {X 0,Y 346.494,Z 281.903,A -85,B 0,C 180,E1 -13937.108,E2 -13937.108} C_VEL
LIN {X 0,Y 346.369,Z 282.34,A -85,B 0,C 180,E1 -13938.293,E2 -13938.293} C_VEL
LIN {X 0,Y 346.226,Z 282.015,A -85,B 0,C 180,E1 -13940.654,E2 -13940.654} C_VEL
LIN {X 0,Y 346.299,Z 281.268,A -85,B 0,C 180,E1 -13941.833,E2 -13941.833} C_VEL
LIN {X 0,Y 346.535,Z 279.343,A -85,B 0,C 180,E1 -13943.595,E2 -13943.595} C_VEL
LIN {X 0,Y 346.694,Z 275.299,A -85,B 0,C 180,E1 -13945.931,E2 -13945.931} C_VEL
LIN {X 0,Y 347.087,Z 271.049,A -85,B 0,C 180,E1 -13947.679,E2 -13947.679} C_VEL
LIN {X 0,Y 347.467,Z 265.644,A -85,B 0,C 180,E1 -13949.421,E2 -13949.421} C_VEL
LIN {X 0,Y 348.22,Z 258.87,A -85,B 0,C 180,E1 -13951.157,E2 -13951.157} C_VEL
LIN {X 0,Y 348.994,Z 250.458,A -85,B 0,C 180,E1 -13952.886,E2 -13952.886} C_VEL
LIN {X 0,Y 349.728,Z 241.824,A -85,B 0,C 180,E1 -13954.322,E2 -13954.322} C_VEL
LIN {X 0,Y 350.845,Z 232.296,A -85,B 0,C 180,E1 -13955.604,E2 -13955.604} C_VEL
LIN {X 0,Y 351.743,Z 221.94,A -85,B 0,C 180,E1 -13956.741,E2 -13956.741} C_VEL
LIN {X 0,Y 352.559,Z 210.578,A -85,B 0,C 180,E1 -13957.733,E2 -13957.733} C_VEL
LIN {X 0,Y 353.182,Z 198.86,A -85,B 0,C 180,E1 -13958.511,E2 -13958.511} C_VEL
LIN {X 0,Y 353.712,Z 185.354,A -85,B 0,C 180,E1 -13959.146,E2 -13959.146} C_VEL
LIN {X 0,Y 354.064,Z 173.25,A -85,B 0,C 180,E1 -13959.497,E2 -13959.497} C_VEL
LIN {X 0,Y 355.249,Z 94.113,A -85,B 0,C 180,E1 -13961.091,E2 -13961.091} C_VEL
LIN {X 0,Y 353.339,Z 86.532,A -85,B 0,C 180,E1 -13961.352,E2 -13961.352} C_VEL
LIN {X 0,Y 348.429,Z 72.005,A -85,B 0,C 180,E1 -13961.935,E2 -13961.935} C_VEL
LIN {X 0,Y 347.878,Z 69.154,A -85,B 0,C 180,E1 -13962.766,E2 -13962.766} C_VEL
LIN {X 0,Y 347.867,Z 69.151,A -85,B 0,C 180,E1 -13965.227,E2 -13965.227} C_VEL
LIN {X 0,Y 347.834,Z 69.157,A -85,B 0,C 180,E1 -13966.656,E2 -13966.656} C_VEL
LIN {X 0,Y 347.147,Z 69.241,A -85,B 0,C 180,E1 -13967.622,E2 -13967.622} C_VEL
LIN {X 0,Y 344.241,Z 69.602,A -85,B 0,C 180,E1 -13969.192,E2 -13969.192} C_VEL
LIN {X 0,Y 341.81,Z 69.909,A -85,B 0,C 180,E1 -13970.464,E2 -13970.464} C_VEL
LIN {X 0,Y 340.804,Z 70.03,A -85,B 0,C 180,E1 -13971.448,E2 -13971.448} C_VEL
LIN {X 0,Y 340.741,Z 70.039,A -85,B 0,C 180,E1 -13971.781,E2 -13971.781} C_VEL
LIN {X 0,Y 340.773,Z 70.035,A -85,B 0,C 180,E1 -13975.665,E2 -13975.665} C_VEL
LIN {X 0,Y 340.73,Z 70.043,A -85,B 0,C 180,E1 -13978.321,E2 -13978.321} C_VEL
LIN {X 0,Y 340.699,Z 70.043,A -85,B 0,C 180,E1 -13981.045,E2 -13981.045} C_VEL
LIN {X 0,Y 340.72,Z 70.042,A -85,B 0,C 180,E1 -13985.279,E2 -13985.279} C_VEL
LIN {X 0,Y 340.714,Z 70.042,A -85,B 0,C 180,E1 -13988.387,E2 -13988.387} C_VEL
LIN {X 0,Y 340.701,Z 70.044,A -85,B 0,C 180,E1 -13992.046,E2 -13992.046} C_VEL
LIN {X 0,Y 340.654,Z 70.049,A -85,B 0,C 180,E1 -13996.227,E2 -13996.227} C_VEL
LIN {X 0,Y 340.69,Z 70.046,A -85,B 0,C 180,E1 -13999.753,E2 -13999.753} C_VEL
LIN {X 0,Y 340.707,Z 70.047,A -85,B 0,C 180,E1 -14003.259,E2 -14003.259} C_VEL
LIN {X 0,Y 340.695,Z 70.043,A -85,B 0,C 180,E1 -14006.154,E2 -14006.154} C_VEL
LIN {X 0,Y 340.744,Z 70.038,A -85,B 0,C 180,E1 -14010.33,E2 -14010.33} C_VEL
LIN {X 0,Y 340.806,Z 70.033,A -85,B 0,C 180,E1 -14013.02,E2 -14013.02} C_VEL
LIN {X 0,Y 340.733,Z 70.042,A -85,B 0,C 180,E1 -14016.928,E2 -14016.928} C_VEL
LIN {X 0,Y 340.794,Z 70.034,A -85,B 0,C 180,E1 -14020.734,E2 -14020.734} C_VEL
LIN {X 0,Y 340.79,Z 70.03,A -85,B 0,C 180,E1 -14023.219,E2 -14023.219} C_VEL
LIN {X 0,Y 340.848,Z 70.025,A -85,B 0,C 180,E1 -14026.891,E2 -14026.891} C_VEL
LIN {X 0,Y 340.888,Z 70.022,A -85,B 0,C 180,E1 -14030.507,E2 -14030.507} C_VEL
LIN {X 0,Y 341.061,Z 69.998,A -85,B 0,C 180,E1 -14032.898,E2 -14032.898} C_VEL
LIN {X 0,Y 341.169,Z 69.986,A -85,B 0,C 180,E1 -14037.639,E2 -14037.639} C_VEL
LIN {X 0,Y 341.3,Z 69.973,A -85,B 0,C 180,E1 -14040,E2 -14040} C_VEL
LIN {X 0,Y 341.172,Z 69.985,A -85,B 0,C 180,E1 -14042.361,E2 -14042.361} C_VEL
LIN {X 0,Y 341.008,Z 70.006,A -85,B 0,C 180,E1 -14047.103,E2 -14047.103} C_VEL
LIN {X 0,Y 340.853,Z 70.024,A -85,B 0,C 180,E1 -14050.695,E2 -14050.695} C_VEL
LIN {X 0,Y 340.867,Z 70.022,A -85,B 0,C 180,E1 -14054.325,E2 -14054.325} C_VEL
LIN {X 0,Y 340.79,Z 70.032,A -85,B 0,C 180,E1 -14058.441,E2 -14058.441} C_VEL
LIN {X 0,Y 340.758,Z 70.036,A -85,B 0,C 180,E1 -14061.857,E2 -14061.857} C_VEL
LIN {X 0,Y 340.749,Z 70.037,A -85,B 0,C 180,E1 -14065.666,E2 -14065.666} C_VEL
LIN {X 0,Y 340.735,Z 70.039,A -85,B 0,C 180,E1 -14069.672,E2 -14069.672} C_VEL
LIN {X 0,Y 340.696,Z 70.044,A -85,B 0,C 180,E1 -14073.847,E2 -14073.847} C_VEL
LIN {X 0,Y 340.708,Z 70.046,A -85,B 0,C 180,E1 -14076.741,E2 -14076.741} C_VEL
LIN {X 0,Y 340.692,Z 70.048,A -85,B 0,C 180,E1 -14080.247,E2 -14080.247} C_VEL
LIN {X 0,Y 340.655,Z 70.05,A -85,B 0,C 180,E1 -14083.773,E2 -14083.773} C_VEL
LIN {X 0,Y 340.699,Z 70.047,A -85,B 0,C 180,E1 -14087.955,E2 -14087.955} C_VEL
LIN {X 0,Y 340.722,Z 70.044,A -85,B 0,C 180,E1 -14091.771,E2 -14091.771} C_VEL
LIN {X 0,Y 340.726,Z 70.043,A -85,B 0,C 180,E1 -14095.595,E2 -14095.595} C_VEL
LIN {X 0,Y 340.746,Z 70.146,A -85,B 0,C 180,E1 -14099.22,E2 -14099.22} C_VEL
LIN {X 0,Y 343.325,Z 82.133,A -85,B 0,C 180,E1 -14102.244,E2 -14102.244} C_VEL
LIN {X 0,Y 344.342,Z 89,A -85,B 0,C 180,E1 -14103.902,E2 -14103.902} C_VEL
LIN {X 0,Y 342.841,Z 104.693,A -85,B 0,C 180,E1 -14107.421,E2 -14107.421} C_VEL
LIN {X 0,Y 342.716,Z 106.106,A -85,B 0,C 180,E1 -14107.737,E2 -14107.737} C_VEL
LIN {X 0,Y 347.781,Z 145.923,A -85,B 0,C 180,E1 -14108.869,E2 -14108.869} C_VEL
LIN {X 0,Y 346.737,Z 214.833,A -85,B 0,C 180,E1 -14110.307,E2 -14110.307} C_VEL
LIN {X 0,Y 346.066,Z 228.223,A -85,B 0,C 180,E1 -14110.807,E2 -14110.807} C_VEL
LIN {X 0,Y 345.141,Z 241.036,A -85,B 0,C 180,E1 -14111.525,E2 -14111.525} C_VEL
LIN {X 0,Y 344.137,Z 253.222,A -85,B 0,C 180,E1 -14112.468,E2 -14112.468} C_VEL
LIN {X 0,Y 343.03,Z 264.823,A -85,B 0,C 180,E1 -14113.637,E2 -14113.637} C_VEL
LIN {X 0,Y 342.012,Z 275.353,A -85,B 0,C 180,E1 -14114.974,E2 -14114.974} C_VEL
LIN {X 0,Y 341.239,Z 283.824,A -85,B 0,C 180,E1 -14116.299,E2 -14116.299} C_VEL
LIN {X 0,Y 340.38,Z 293.067,A -85,B 0,C 180,E1 -14118.084,E2 -14118.084} C_VEL
LIN {X 0,Y 339.72,Z 300.5,A -85,B 0,C 180,E1 -14119.872,E2 -14119.872} C_VEL
LIN {X 0,Y 339.392,Z 306.463,A -85,B 0,C 180,E1 -14121.665,E2 -14121.665} C_VEL
LIN {X 0,Y 339.143,Z 311.147,A -85,B 0,C 180,E1 -14123.455,E2 -14123.455} C_VEL
LIN {X 0,Y 339.185,Z 314.71,A -85,B 0,C 180,E1 -14125.246,E2 -14125.246} C_VEL
LIN {X 0,Y 339.171,Z 316.504,A -85,B 0,C 180,E1 -14126.436,E2 -14126.436} C_VEL
LIN {X 0,Y 339.221,Z 317.857,A -85,B 0,C 180,E1 -14127.625,E2 -14127.625} C_VEL
LIN {X 0,Y 339.329,Z 318.81,A -85,B 0,C 180,E1 -14128.813,E2 -14128.813} C_VEL
LIN {X 0,Y 339.331,Z 319.363,A -85,B 0,C 180,E1 -14130,E2 -14130} C_VEL
LIN {X 0,Y 339.255,Z 319.479,A -85,B 0,C 180,E1 -14131.187,E2 -14131.187} C_VEL
LIN {X 0,Y 339.114,Z 318.51,A -85,B 0,C 180,E1 -14133.565,E2 -14133.565} C_VEL
LIN {X 0,Y 339.082,Z 316.163,A -85,B 0,C 180,E1 -14135.801,E2 -14135.801} C_VEL
LIN {X 0,Y 339.324,Z 312.91,A -85,B 0,C 180,E1 -14137.737,E2 -14137.737} C_VEL
LIN {X 0,Y 339.691,Z 308.834,A -85,B 0,C 180,E1 -14139.527,E2 -14139.527} C_VEL
LIN {X 0,Y 340.428,Z 302.607,A -85,B 0,C 180,E1 -14141.612,E2 -14141.612} C_VEL
LIN {X 0,Y 341.555,Z 295.861,A -85,B 0,C 180,E1 -14143.385,E2 -14143.385} C_VEL
LIN {X 0,Y 342.787,Z 287.523,A -85,B 0,C 180,E1 -14145.154,E2 -14145.154} C_VEL
LIN {X 0,Y 344.067,Z 278.98,A -85,B 0,C 180,E1 -14146.617,E2 -14146.617} C_VEL
LIN {X 0,Y 345.692,Z 268.47,A -85,B 0,C 180,E1 -14148.061,E2 -14148.061} C_VEL
LIN {X 0,Y 347.428,Z 256.659,A -85,B 0,C 180,E1 -14149.344,E2 -14149.344} C_VEL
LIN {X 0,Y 348.851,Z 244.779,A -85,B 0,C 180,E1 -14150.336,E2 -14150.336} C_VEL
LIN {X 0,Y 350.163,Z 232.439,A -85,B 0,C 180,E1 -14151.101,E2 -14151.101} C_VEL
LIN {X 0,Y 351.136,Z 219.776,A -85,B 0,C 180,E1 -14151.656,E2 -14151.656} C_VEL
LIN {X 0,Y 351.678,Z 206.564,A -85,B 0,C 180,E1 -14152.006,E2 -14152.006} C_VEL
LIN {X 0,Y 352.828,Z 146.54,A -85,B 0,C 180,E1 -14153.253,E2 -14153.253} C_VEL
LIN {X 0,Y 348.902,Z 122.781,A -85,B 0,C 180,E1 -14154.112,E2 -14154.112} C_VEL
LIN {X 0,Y 345.357,Z 105.267,A -85,B 0,C 180,E1 -14154.838,E2 -14154.838} C_VEL
LIN {X 0,Y 346.425,Z 96.866,A -85,B 0,C 180,E1 -14156.793,E2 -14156.793} C_VEL
LIN {X 0,Y 346.046,Z 92.702,A -85,B 0,C 180,E1 -14157.847,E2 -14157.847} C_VEL
LIN {X 0,Y 343.372,Z 80.704,A -85,B 0,C 180,E1 -14161.118,E2 -14161.118} C_VEL
LIN {X 0,Y 340.725,Z 70.043,A -85,B 0,C 180,E1 -14164.207,E2 -14164.207} C_VEL
LIN {X 0,Y 340.735,Z 70.038,A -85,B 0,C 180,E1 -14168.227,E2 -14168.227} C_VEL
LIN {X 0,Y 340.701,Z 70.042,A -85,B 0,C 180,E1 -14172.045,E2 -14172.045} C_VEL
LIN {X 0,Y 340.654,Z 70.047,A -85,B 0,C 180,E1 -14176.227,E2 -14176.227} C_VEL
LIN {X 0,Y 340.69,Z 70.039,A -85,B 0,C 180,E1 -14179.753,E2 -14179.753} C_VEL
LIN {X 0,Y 340.707,Z 70.038,A -85,B 0,C 180,E1 -14183.258,E2 -14183.258} C_VEL
LIN {X 0,Y 340.695,Z 70.039,A -85,B 0,C 180,E1 -14186.153,E2 -14186.153} C_VEL
LIN {X 0,Y 340.777,Z 70.029,A -85,B 0,C 180,E1 -14190.332,E2 -14190.332} C_VEL
LIN {X 0,Y 340.808,Z 70.03,A -85,B 0,C 180,E1 -14193.02,E2 -14193.02} C_VEL
LIN {X 0,Y 340.732,Z 70.04,A -85,B 0,C 180,E1 -14196.927,E2 -14196.927} C_VEL
LIN {X 0,Y 340.794,Z 70.035,A -85,B 0,C 180,E1 -14200.734,E2 -14200.734} C_VEL
LIN {X 0,Y 340.79,Z 70.026,A -85,B 0,C 180,E1 -14203.219,E2 -14203.219} C_VEL
LIN {X 0,Y 340.847,Z 70.02,A -85,B 0,C 180,E1 -14206.89,E2 -14206.89} C_VEL
LIN {X 0,Y 340.917,Z 70.02,A -85,B 0,C 180,E1 -14210.507,E2 -14210.507} C_VEL
LIN {X 0,Y 341.062,Z 69.988,A -85,B 0,C 180,E1 -14212.898,E2 -14212.898} C_VEL
LIN {X 0,Y 341.169,Z 69.981,A -85,B 0,C 180,E1 -14217.639,E2 -14217.639} C_VEL
LIN {X 0,Y 341.298,Z 69.97,A -85,B 0,C 180,E1 -14220,E2 -14220} C_VEL
LIN {X 0,Y 341.17,Z 69.982,A -85,B 0,C 180,E1 -14222.361,E2 -14222.361} C_VEL
LIN {X 0,Y 341.048,Z 70.003,A -85,B 0,C 180,E1 -14227.102,E2 -14227.102} C_VEL
LIN {X 0,Y 340.851,Z 70.024,A -85,B 0,C 180,E1 -14230.694,E2 -14230.694} C_VEL
LIN {X 0,Y 340.866,Z 70.015,A -85,B 0,C 180,E1 -14234.325,E2 -14234.325} C_VEL
LIN {X 0,Y 340.789,Z 70.027,A -85,B 0,C 180,E1 -14238.441,E2 -14238.441} C_VEL
LIN {X 0,Y 340.756,Z 70.036,A -85,B 0,C 180,E1 -14241.857,E2 -14241.857} C_VEL
LIN {X 0,Y 340.748,Z 70.038,A -85,B 0,C 180,E1 -14245.666,E2 -14245.666} C_VEL
LIN {X 0,Y 340.733,Z 70.04,A -85,B 0,C 180,E1 -14249.671,E2 -14249.671} C_VEL
LIN {X 0,Y 340.694,Z 70.043,A -85,B 0,C 180,E1 -14253.846,E2 -14253.846} C_VEL
LIN {X 0,Y 340.704,Z 70.042,A -85,B 0,C 180,E1 -14256.742,E2 -14256.742} C_VEL
LIN {X 0,Y 340.674,Z 70.036,A -85,B 0,C 180,E1 -14260.244,E2 -14260.244} C_VEL
LIN {X 0,Y 340.653,Z 70.055,A -85,B 0,C 180,E1 -14263.773,E2 -14263.773} C_VEL
LIN {X 0,Y 340.699,Z 70.047,A -85,B 0,C 180,E1 -14267.955,E2 -14267.955} C_VEL
LIN {X 0,Y 340.72,Z 70.046,A -85,B 0,C 180,E1 -14271.771,E2 -14271.771} C_VEL
LIN {X 0,Y 340.723,Z 70.083,A -85,B 0,C 180,E1 -14273.778,E2 -14273.778} C_VEL
LIN {X 0,Y 341.531,Z 73.286,A -85,B 0,C 180,E1 -14274.856,E2 -14274.856} C_VEL
LIN {X 0,Y 350.979,Z 94.03,A -85,B 0,C 180,E1 -14276.198,E2 -14276.198} C_VEL
LIN {X 0,Y 353.982,Z 101.781,A -85,B 0,C 180,E1 -14276.627,E2 -14276.627} C_VEL
LIN {X 0,Y 351.992,Z 180.47,A -85,B 0,C 180,E1 -14278.265,E2 -14278.265} C_VEL
LIN {X 0,Y 351.358,Z 194.245,A -85,B 0,C 180,E1 -14278.812,E2 -14278.812} C_VEL
LIN {X 0,Y 350.621,Z 206.361,A -85,B 0,C 180,E1 -14279.532,E2 -14279.532} C_VEL
LIN {X 0,Y 349.468,Z 218.304,A -85,B 0,C 180,E1 -14280.481,E2 -14280.481} C_VEL
LIN {X 0,Y 348.002,Z 229.92,A -85,B 0,C 180,E1 -14281.667,E2 -14281.667} C_VEL
LIN {X 0,Y 346.524,Z 240.51,A -85,B 0,C 180,E1 -14283.047,E2 -14283.047} C_VEL
LIN {X 0,Y 345.009,Z 250.398,A -85,B 0,C 180,E1 -14284.673,E2 -14284.673} C_VEL
LIN {X 0,Y 343.774,Z 257.855,A -85,B 0,C 180,E1 -14286.186,E2 -14286.186} C_VEL
LIN {X 0,Y 342.678,Z 264.201,A -85,B 0,C 180,E1 -14287.756,E2 -14287.756} C_VEL
LIN {X 0,Y 341.624,Z 270,A -85,B 0,C 180,E1 -14289.529,E2 -14289.529} C_VEL
LIN {X 0,Y 340.76,Z 275.144,A -85,B 0,C 180,E1 -14291.573,E2 -14291.573} C_VEL
LIN {X 0,Y 340.192,Z 278.211,A -85,B 0,C 180,E1 -14293.188,E2 -14293.188} C_VEL
LIN {X 0,Y 339.84,Z 279.968,A -85,B 0,C 180,E1 -14294.404,E2 -14294.404} C_VEL
LIN {X 0,Y 339.464,Z 282.089,A -85,B 0,C 180,E1 -14296.668,E2 -14296.668} C_VEL
LIN {X 0,Y 339.298,Z 282.707,A -85,B 0,C 180,E1 -14298.046,E2 -14298.046} C_VEL
LIN {X 0,Y 339.142,Z 282.459,A -85,B 0,C 180,E1 -14300.457,E2 -14300.457} C_VEL
LIN {X 0,Y 339.197,Z 281.752,A -85,B 0,C 180,E1 -14301.661,E2 -14301.661} C_VEL
LIN {X 0,Y 339.46,Z 279.729,A -85,B 0,C 180,E1 -14303.599,E2 -14303.599} C_VEL
LIN {X 0,Y 339.593,Z 275.975,A -85,B 0,C 180,E1 -14305.846,E2 -14305.846} C_VEL
LIN {X 0,Y 339.99,Z 271.811,A -85,B 0,C 180,E1 -14307.631,E2 -14307.631} C_VEL
LIN {X 0,Y 340.478,Z 265.495,A -85,B 0,C 180,E1 -14309.704,E2 -14309.704} C_VEL
LIN {X 0,Y 341.263,Z 258.598,A -85,B 0,C 180,E1 -14311.475,E2 -14311.475} C_VEL
LIN {X 0,Y 342.079,Z 249.981,A -85,B 0,C 180,E1 -14313.239,E2 -14313.239} C_VEL
LIN {X 0,Y 342.923,Z 241.162,A -85,B 0,C 180,E1 -14314.702,E2 -14314.702} C_VEL
LIN {X 0,Y 344.011,Z 231.436,A -85,B 0,C 180,E1 -14316.01,E2 -14316.01} C_VEL
LIN {X 0,Y 344.982,Z 220.779,A -85,B 0,C 180,E1 -14317.168,E2 -14317.168} C_VEL
LIN {X 0,Y 345.812,Z 208.865,A -85,B 0,C 180,E1 -14318.179,E2 -14318.179} C_VEL
LIN {X 0,Y 346.503,Z 196.46,A -85,B 0,C 180,E1 -14318.97,E2 -14318.97} C_VEL
LIN {X 0,Y 346.988,Z 184.515,A -85,B 0,C 180,E1 -14319.509,E2 -14319.509} C_VEL
LIN {X 0,Y 347.303,Z 169.654,A -85,B 0,C 180,E1 -14319.905,E2 -14319.905} C_VEL
LIN {X 0,Y 348.446,Z 94.693,A -85,B 0,C 180,E1 -14321.444,E2 -14321.444} C_VEL
LIN {X 0,Y 345.955,Z 86.101,A -85,B 0,C 180,E1 -14321.767,E2 -14321.767} C_VEL
LIN {X 0,Y 341.286,Z 72.388,A -85,B 0,C 180,E1 -14322.336,E2 -14322.336} C_VEL
LIN {X 0,Y 340.853,Z 70.029,A -85,B 0,C 180,E1 -14323.034,E2 -14323.034} C_VEL
LIN {X 0,Y 340.785,Z 70.034,A -85,B 0,C 180,E1 -14326.661,E2 -14326.661} C_VEL
LIN {X 0,Y 340.794,Z 70.031,A -85,B 0,C 180,E1 -14329.267,E2 -14329.267} C_VEL
LIN {X 0,Y 340.741,Z 70.039,A -85,B 0,C 180,E1 -14331.781,E2 -14331.781} C_VEL
LIN {X 0,Y 340.122,Z 70.12,A -85,B 0,C 180,E1 -14332.769,E2 -14332.769} C_VEL
LIN {X 0,Y 337.273,Z 70.476,A -85,B 0,C 180,E1 -14334.374,E2 -14334.374} C_VEL
LIN {X 0,Y 334.834,Z 70.777,A -85,B 0,C 180,E1 -14335.675,E2 -14335.675} C_VEL
LIN {X 0,Y 333.795,Z 70.905,A -85,B 0,C 180,E1 -14336.682,E2 -14336.682} C_VEL
LIN {X 0,Y 333.717,Z 70.913,A -85,B 0,C 180,E1 -14337.023,E2 -14337.023} C_VEL
LIN {X 0,Y 333.692,Z 70.918,A -85,B 0,C 180,E1 -14340.363,E2 -14340.363} C_VEL
LIN {X 0,Y 333.676,Z 70.918,A -85,B 0,C 180,E1 -14344.659,E2 -14344.659} C_VEL
LIN {X 0,Y 333.656,Z 70.925,A -85,B 0,C 180,E1 -14347.651,E2 -14347.651} C_VEL
LIN {X 0,Y 333.648,Z 70.921,A -85,B 0,C 180,E1 -14350.768,E2 -14350.768} C_VEL
LIN {X 0,Y 333.595,Z 70.928,A -85,B 0,C 180,E1 -14354.251,E2 -14354.251} C_VEL
LIN {X 0,Y 333.644,Z 70.925,A -85,B 0,C 180,E1 -14357.619,E2 -14357.619} C_VEL
LIN {X 0,Y 333.655,Z 70.925,A -85,B 0,C 180,E1 -14361.202,E2 -14361.202} C_VEL
LIN {X 0,Y 333.679,Z 70.917,A -85,B 0,C 180,E1 -14363.861,E2 -14363.861} C_VEL
LIN {X 0,Y 333.646,Z 70.924,A -85,B 0,C 180,E1 -14367.413,E2 -14367.413} C_VEL
LIN {X 0,Y 333.693,Z 70.92,A -85,B 0,C 180,E1 -14371.026,E2 -14371.026} C_VEL
LIN {X 0,Y 333.738,Z 70.91,A -85,B 0,C 180,E1 -14373.754,E2 -14373.754} C_VEL
LIN {X 0,Y 333.723,Z 70.912,A -85,B 0,C 180,E1 -14377.914,E2 -14377.914} C_VEL
LIN {X 0,Y 333.797,Z 70.902,A -85,B 0,C 180,E1 -14381.59,E2 -14381.59} C_VEL
LIN {X 0,Y 333.812,Z 70.9,A -85,B 0,C 180,E1 -14385.577,E2 -14385.577} C_VEL
LIN {X 0,Y 333.822,Z 70.9,A -85,B 0,C 180,E1 -14389.078,E2 -14389.078} C_VEL
LIN {X 0,Y 334.008,Z 70.876,A -85,B 0,C 180,E1 -14392.747,E2 -14392.747} C_VEL
LIN {X 0,Y 333.806,Z 70.899,A -85,B 0,C 180,E1 -14395.169,E2 -14395.169} C_VEL
LIN {X 0,Y 334.107,Z 70.865,A -85,B 0,C 180,E1 -14397.589,E2 -14397.589} C_VEL
LIN {X 0,Y 334.25,Z 70.851,A -85,B 0,C 180,E1 -14400,E2 -14400} C_VEL
LIN {X 0,Y 334.109,Z 70.865,A -85,B 0,C 180,E1 -14402.411,E2 -14402.411} C_VEL
LIN {X 0,Y 333.996,Z 70.88,A -85,B 0,C 180,E1 -14406.039,E2 -14406.039} C_VEL
LIN {X 0,Y 333.825,Z 70.903,A -85,B 0,C 180,E1 -14409.696,E2 -14409.696} C_VEL
LIN {X 0,Y 333.801,Z 70.908,A -85,B 0,C 180,E1 -14413.391,E2 -14413.391} C_VEL
LIN {X 0,Y 333.724,Z 70.917,A -85,B 0,C 180,E1 -14417.148,E2 -14417.148} C_VEL
LIN {X 0,Y 333.724,Z 70.913,A -85,B 0,C 180,E1 -14419.691,E2 -14419.691} C_VEL
LIN {X 0,Y 333.696,Z 70.916,A -85,B 0,C 180,E1 -14422.278,E2 -14422.278} C_VEL
LIN {X 0,Y 333.71,Z 70.918,A -85,B 0,C 180,E1 -14425.096,E2 -14425.096} C_VEL
LIN {X 0,Y 333.674,Z 70.923,A -85,B 0,C 180,E1 -14428.976,E2 -14428.976} C_VEL
LIN {X 0,Y 333.647,Z 70.927,A -85,B 0,C 180,E1 -14432.587,E2 -14432.587} C_VEL
LIN {X 0,Y 333.679,Z 70.92,A -85,B 0,C 180,E1 -14436.139,E2 -14436.139} C_VEL
LIN {X 0,Y 333.65,Z 70.922,A -85,B 0,C 180,E1 -14439.192,E2 -14439.192} C_VEL
LIN {X 0,Y 333.636,Z 70.927,A -85,B 0,C 180,E1 -14442.5,E2 -14442.5} C_VEL
LIN {X 0,Y 333.599,Z 70.931,A -85,B 0,C 180,E1 -14445.955,E2 -14445.955} C_VEL
LIN {X 0,Y 333.645,Z 70.923,A -85,B 0,C 180,E1 -14449.316,E2 -14449.316} C_VEL
LIN {X 0,Y 333.666,Z 70.92,A -85,B 0,C 180,E1 -14453.168,E2 -14453.168} C_VEL
LIN {X 0,Y 333.677,Z 70.92,A -85,B 0,C 180,E1 -14455.341,E2 -14455.341} C_VEL
LIN {X 0,Y 333.701,Z 70.957,A -85,B 0,C 180,E1 -14458.893,E2 -14458.893} C_VEL
LIN {X 0,Y 336.547,Z 84.318,A -85,B 0,C 180,E1 -14462.334,E2 -14462.334} C_VEL
LIN {X 0,Y 337.391,Z 89.431,A -85,B 0,C 180,E1 -14463.6,E2 -14463.6} C_VEL
LIN {X 0,Y 335.999,Z 104.138,A -85,B 0,C 180,E1 -14466.976,E2 -14466.976} C_VEL
LIN {X 0,Y 335.824,Z 105.741,A -85,B 0,C 180,E1 -14467.341,E2 -14467.341} C_VEL
LIN {X 0,Y 340.878,Z 145.177,A -85,B 0,C 180,E1 -14468.491,E2 -14468.491} C_VEL
LIN {X 0,Y 340.473,Z 182.9,A -85,B 0,C 180,E1 -14469.289,E2 -14469.289} C_VEL
LIN {X 0,Y 339.879,Z 215.676,A -85,B 0,C 180,E1 -14470.011,E2 -14470.011} C_VEL
LIN {X 0,Y 339.155,Z 229.428,A -85,B 0,C 180,E1 -14470.558,E2 -14470.558} C_VEL
LIN {X 0,Y 338.201,Z 241.773,A -85,B 0,C 180,E1 -14471.288,E2 -14471.288} C_VEL
LIN {X 0,Y 337.177,Z 253.665,A -85,B 0,C 180,E1 -14472.251,E2 -14472.251} C_VEL
LIN {X 0,Y 336.04,Z 265.115,A -85,B 0,C 180,E1 -14473.444,E2 -14473.444} C_VEL
LIN {X 0,Y 335.008,Z 275.458,A -85,B 0,C 180,E1 -14474.801,E2 -14474.801} C_VEL
LIN {X 0,Y 334.092,Z 284.705,A -85,B 0,C 180,E1 -14476.311,E2 -14476.311} C_VEL
LIN {X 0,Y 333.236,Z 293.73,A -85,B 0,C 180,E1 -14478.133,E2 -14478.133} C_VEL
LIN {X 0,Y 332.598,Z 300.972,A -85,B 0,C 180,E1 -14479.96,E2 -14479.96} C_VEL
LIN {X 0,Y 332.32,Z 305.864,A -85,B 0,C 180,E1 -14481.487,E2 -14481.487} C_VEL
LIN {X 0,Y 332.064,Z 310.595,A -85,B 0,C 180,E1 -14483.315,E2 -14483.315} C_VEL
LIN {X 0,Y 332.091,Z 314.201,A -85,B 0,C 180,E1 -14485.144,E2 -14485.144} C_VEL
LIN {X 0,Y 332.093,Z 316.036,A -85,B 0,C 180,E1 -14486.36,E2 -14486.36} C_VEL
LIN {X 0,Y 332.233,Z 318.379,A -85,B 0,C 180,E1 -14488.788,E2 -14488.788} C_VEL
LIN {X 0,Y 332.27,Z 318.952,A -85,B 0,C 180,E1 -14490,E2 -14490} C_VEL
LIN {X 0,Y 332.158,Z 319.103,A -85,B 0,C 180,E1 -14491.212,E2 -14491.212} C_VEL
LIN {X 0,Y 332.035,Z 318.17,A -85,B 0,C 180,E1 -14493.641,E2 -14493.641} C_VEL
LIN {X 0,Y 332.005,Z 316.043,A -85,B 0,C 180,E1 -14495.78,E2 -14495.78} C_VEL
LIN {X 0,Y 332.247,Z 312.66,A -85,B 0,C 180,E1 -14497.903,E2 -14497.903} C_VEL
LIN {X 0,Y 332.651,Z 308.626,A -85,B 0,C 180,E1 -14499.731,E2 -14499.731} C_VEL
LIN {X 0,Y 333.428,Z 302.46,A -85,B 0,C 180,E1 -14501.859,E2 -14501.859} C_VEL
LIN {X 0,Y 334.641,Z 295.769,A -85,B 0,C 180,E1 -14503.666,E2 -14503.666} C_VEL
LIN {X 0,Y 335.932,Z 287.494,A -85,B 0,C 180,E1 -14505.47,E2 -14505.47} C_VEL
LIN {X 0,Y 337.255,Z 279.047,A -85,B 0,C 180,E1 -14506.962,E2 -14506.962} C_VEL
LIN {X 0,Y 338.953,Z 268.645,A -85,B 0,C 180,E1 -14508.433,E2 -14508.433} C_VEL
LIN {X 0,Y 340.741,Z 256.962,A -85,B 0,C 180,E1 -14509.74,E2 -14509.74} C_VEL
LIN {X 0,Y 342.245,Z 245.343,A -85,B 0,C 180,E1 -14510.746,E2 -14510.746} C_VEL
LIN {X 0,Y 343.592,Z 233.295,A -85,B 0,C 180,E1 -14511.525,E2 -14511.525} C_VEL
LIN {X 0,Y 344.647,Z 220.237,A -85,B 0,C 180,E1 -14512.124,E2 -14512.124} C_VEL
LIN {X 0,Y 345.248,Z 207.801,A -85,B 0,C 180,E1 -14512.477,E2 -14512.477} C_VEL
LIN {X 0,Y 346.486,Z 147.498,A -85,B 0,C 180,E1 -14513.751,E2 -14513.751} C_VEL
LIN {X 0,Y 342.779,Z 124.841,A -85,B 0,C 180,E1 -14514.594,E2 -14514.594} C_VEL
LIN {X 0,Y 338.727,Z 104.797,A -85,B 0,C 180,E1 -14515.464,E2 -14515.464} C_VEL
LIN {X 0,Y 339.589,Z 96.66,A -85,B 0,C 180,E1 -14517.417,E2 -14517.417} C_VEL
LIN {X 0,Y 337.609,Z 87.319,A -85,B 0,C 180,E1 -14519.974,E2 -14519.974} C_VEL
LIN {X 0,Y 335.14,Z 76.687,A -85,B 0,C 180,E1 -14523.041,E2 -14523.041} C_VEL
LIN {X 0,Y 333.668,Z 70.922,A -85,B 0,C 180,E1 -14524.849,E2 -14524.849} C_VEL
LIN {X 0,Y 333.654,Z 70.926,A -85,B 0,C 180,E1 -14527.651,E2 -14527.651} C_VEL
LIN {X 0,Y 333.649,Z 70.922,A -85,B 0,C 180,E1 -14530.767,E2 -14530.767} C_VEL
LIN {X 0,Y 333.596,Z 70.925,A -85,B 0,C 180,E1 -14534.25,E2 -14534.25} C_VEL
LIN {X 0,Y 333.644,Z 70.918,A -85,B 0,C 180,E1 -14537.619,E2 -14537.619} C_VEL
LIN {X 0,Y 333.655,Z 70.918,A -85,B 0,C 180,E1 -14541.202,E2 -14541.202} C_VEL
LIN {X 0,Y 333.678,Z 70.916,A -85,B 0,C 180,E1 -14543.861,E2 -14543.861} C_VEL
LIN {X 0,Y 333.646,Z 70.922,A -85,B 0,C 180,E1 -14547.413,E2 -14547.413} C_VEL
LIN {X 0,Y 333.714,Z 70.913,A -85,B 0,C 180,E1 -14551.028,E2 -14551.028} C_VEL
LIN {X 0,Y 333.739,Z 70.905,A -85,B 0,C 180,E1 -14553.754,E2 -14553.754} C_VEL
LIN {X 0,Y 333.722,Z 70.909,A -85,B 0,C 180,E1 -14557.914,E2 -14557.914} C_VEL
LIN {X 0,Y 333.797,Z 70.902,A -85,B 0,C 180,E1 -14561.589,E2 -14561.589} C_VEL
LIN {X 0,Y 333.811,Z 70.903,A -85,B 0,C 180,E1 -14565.576,E2 -14565.576} C_VEL
LIN {X 0,Y 333.837,Z 70.897,A -85,B 0,C 180,E1 -14569.078,E2 -14569.078} C_VEL
LIN {X 0,Y 334.009,Z 70.867,A -85,B 0,C 180,E1 -14572.747,E2 -14572.747} C_VEL
LIN {X 0,Y 333.807,Z 70.902,A -85,B 0,C 180,E1 -14575.169,E2 -14575.169} C_VEL
LIN {X 0,Y 334.106,Z 70.861,A -85,B 0,C 180,E1 -14577.589,E2 -14577.589} C_VEL
LIN {X 0,Y 334.249,Z 70.848,A -85,B 0,C 180,E1 -14580,E2 -14580} C_VEL
LIN {X 0,Y 334.107,Z 70.861,A -85,B 0,C 180,E1 -14582.411,E2 -14582.411} C_VEL
LIN {X 0,Y 333.984,Z 70.88,A -85,B 0,C 180,E1 -14586.597,E2 -14586.597} C_VEL
LIN {X 0,Y 333.824,Z 70.896,A -85,B 0,C 180,E1 -14589.696,E2 -14589.696} C_VEL
LIN {X 0,Y 333.8,Z 70.897,A -85,B 0,C 180,E1 -14593.391,E2 -14593.391} C_VEL
LIN {X 0,Y 333.722,Z 70.914,A -85,B 0,C 180,E1 -14597.147,E2 -14597.147} C_VEL
LIN {X 0,Y 333.727,Z 70.912,A -85,B 0,C 180,E1 -14599.691,E2 -14599.691} C_VEL
LIN {X 0,Y 333.694,Z 70.916,A -85,B 0,C 180,E1 -14602.278,E2 -14602.278} C_VEL
LIN {X 0,Y 333.709,Z 70.918,A -85,B 0,C 180,E1 -14605.096,E2 -14605.096} C_VEL
LIN {X 0,Y 333.672,Z 70.922,A -85,B 0,C 180,E1 -14608.976,E2 -14608.976} C_VEL
LIN {X 0,Y 333.645,Z 70.926,A -85,B 0,C 180,E1 -14612.587,E2 -14612.587} C_VEL
LIN {X 0,Y 333.676,Z 70.922,A -85,B 0,C 180,E1 -14616.139,E2 -14616.139} C_VEL
LIN {X 0,Y 333.633,Z 70.925,A -85,B 0,C 180,E1 -14619.194,E2 -14619.194} C_VEL
LIN {X 0,Y 333.632,Z 70.925,A -85,B 0,C 180,E1 -14622.499,E2 -14622.499} C_VEL
LIN {X 0,Y 333.597,Z 70.932,A -85,B 0,C 180,E1 -14625.955,E2 -14625.955} C_VEL
LIN {X 0,Y 333.644,Z 70.926,A -85,B 0,C 180,E1 -14629.316,E2 -14629.316} C_VEL
LIN {X 0,Y 333.676,Z 71.011,A -85,B 0,C 180,E1 -14633.247,E2 -14633.247} C_VEL
LIN {X 0,Y 334.395,Z 73.879,A -85,B 0,C 180,E1 -14634.201,E2 -14634.201} C_VEL
LIN {X 0,Y 343.449,Z 93.197,A -85,B 0,C 180,E1 -14635.515,E2 -14635.515} C_VEL
LIN {X 0,Y 347.617,Z 103.241,A -85,B 0,C 180,E1 -14636.118,E2 -14636.118} C_VEL
LIN {X 0,Y 345.609,Z 180.779,A -85,B 0,C 180,E1 -14637.762,E2 -14637.762} C_VEL
LIN {X 0,Y 344.938,Z 194.477,A -85,B 0,C 180,E1 -14638.313,E2 -14638.313} C_VEL
LIN {X 0,Y 344.15,Z 206.83,A -85,B 0,C 180,E1 -14639.059,E2 -14639.059} C_VEL
LIN {X 0,Y 342.945,Z 218.823,A -85,B 0,C 180,E1 -14640.032,E2 -14640.032} C_VEL
LIN {X 0,Y 341.413,Z 230.409,A -85,B 0,C 180,E1 -14641.238,E2 -14641.238} C_VEL
LIN {X 0,Y 339.87,Z 240.963,A -85,B 0,C 180,E1 -14642.64,E2 -14642.64} C_VEL
LIN {X 0,Y 338.402,Z 250.018,A -85,B 0,C 180,E1 -14644.143,E2 -14644.143} C_VEL
LIN {X 0,Y 336.871,Z 258.984,A -85,B 0,C 180,E1 -14645.995,E2 -14645.995} C_VEL
LIN {X 0,Y 335.567,Z 266.076,A -85,B 0,C 180,E1 -14647.853,E2 -14647.853} C_VEL
LIN {X 0,Y 334.482,Z 271.692,A -85,B 0,C 180,E1 -14649.715,E2 -14649.715} C_VEL
LIN {X 0,Y 333.686,Z 276.059,A -85,B 0,C 180,E1 -14651.583,E2 -14651.583} C_VEL
LIN {X 0,Y 333.25,Z 278.352,A -85,B 0,C 180,E1 -14652.827,E2 -14652.827} C_VEL
LIN {X 0,Y 332.865,Z 280.187,A -85,B 0,C 180,E1 -14654.069,E2 -14654.069} C_VEL
LIN {X 0,Y 332.562,Z 281.543,A -85,B 0,C 180,E1 -14655.31,E2 -14655.31} C_VEL
LIN {X 0,Y 332.403,Z 282.493,A -85,B 0,C 180,E1 -14656.551,E2 -14656.551} C_VEL
LIN {X 0,Y 332.23,Z 283.052,A -85,B 0,C 180,E1 -14657.787,E2 -14657.787} C_VEL
LIN {X 0,Y 332.095,Z 283.186,A -85,B 0,C 180,E1 -14659.02,E2 -14659.02} C_VEL
LIN {X 0,Y 332.115,Z 282.231,A -85,B 0,C 180,E1 -14661.482,E2 -14661.482} C_VEL
LIN {X 0,Y 332.378,Z 280.099,A -85,B 0,C 180,E1 -14663.614,E2 -14663.614} C_VEL
LIN {X 0,Y 332.499,Z 276.644,A -85,B 0,C 180,E1 -14665.757,E2 -14665.757} C_VEL
LIN {X 0,Y 332.897,Z 272.564,A -85,B 0,C 180,E1 -14667.58,E2 -14667.58} C_VEL
LIN {X 0,Y 333.402,Z 266.337,A -85,B 0,C 180,E1 -14669.698,E2 -14669.698} C_VEL
LIN {X 0,Y 334.204,Z 259.546,A -85,B 0,C 180,E1 -14671.506,E2 -14671.506} C_VEL
LIN {X 0,Y 335.046,Z 251.102,A -85,B 0,C 180,E1 -14673.307,E2 -14673.307} C_VEL
LIN {X 0,Y 335.874,Z 242.436,A -85,B 0,C 180,E1 -14674.801,E2 -14674.801} C_VEL
LIN {X 0,Y 337.043,Z 232.879,A -85,B 0,C 180,E1 -14676.135,E2 -14676.135} C_VEL
LIN {X 0,Y 338.01,Z 222.48,A -85,B 0,C 180,E1 -14677.317,E2 -14677.317} C_VEL
LIN {X 0,Y 338.886,Z 211.042,A -85,B 0,C 180,E1 -14678.347,E2 -14678.347} C_VEL
LIN {X 0,Y 339.563,Z 199.209,A -85,B 0,C 180,E1 -14679.155,E2 -14679.155} C_VEL
LIN {X 0,Y 340.101,Z 186.438,A -85,B 0,C 180,E1 -14679.778,E2 -14679.778} C_VEL
LIN {X 0,Y 340.5,Z 172.959,A -85,B 0,C 180,E1 -14680.18,E2 -14680.18} C_VEL
LIN {X 0,Y 341.757,Z 95.818,A -85,B 0,C 180,E1 -14681.793,E2 -14681.793} C_VEL
LIN {X 0,Y 336.411,Z 79.183,A -85,B 0,C 180,E1 -14682.471,E2 -14682.471} C_VEL
LIN {X 0,Y 334.149,Z 72.741,A -85,B 0,C 180,E1 -14682.759,E2 -14682.759} C_VEL
LIN {X 0,Y 333.819,Z 70.905,A -85,B 0,C 180,E1 -14683.313,E2 -14683.313} C_VEL
LIN {X 0,Y 333.748,Z 70.91,A -85,B 0,C 180,E1 -14687.146,E2 -14687.146} C_VEL
LIN {X 0,Y 333.737,Z 70.911,A -85,B 0,C 180,E1 -14689.691,E2 -14689.691} C_VEL
LIN {X 0,Y 333.671,Z 70.919,A -85,B 0,C 180,E1 -14693.59,E2 -14693.59} C_VEL
LIN {X 0,Y 333.717,Z 70.913,A -85,B 0,C 180,E1 -14697.023,E2 -14697.023} C_VEL
LIN {X 0,Y 333.046,Z 71.002,A -85,B 0,C 180,E1 -14698.031,E2 -14698.031} C_VEL
LIN {X 0,Y 330.129,Z 71.362,A -85,B 0,C 180,E1 -14699.668,E2 -14699.668} C_VEL
LIN {X 0,Y 327.675,Z 71.665,A -85,B 0,C 180,E1 -14700.996,E2 -14700.996} C_VEL
LIN {X 0,Y 326.66,Z 71.797,A -85,B 0,C 180,E1 -14702.024,E2 -14702.024} C_VEL
LIN {X 0,Y 326.598,Z 71.799,A -85,B 0,C 180,E1 -14702.373,E2 -14702.373} C_VEL
LIN {X 0,Y 326.615,Z 71.8,A -85,B 0,C 180,E1 -14705.52,E2 -14705.52} C_VEL
LIN {X 0,Y 326.614,Z 71.799,A -85,B 0,C 180,E1 -14709.228,E2 -14709.228} C_VEL
LIN {X 0,Y 326.578,Z 71.803,A -85,B 0,C 180,E1 -14712.972,E2 -14712.972} C_VEL
LIN {X 0,Y 326.578,Z 71.804,A -85,B 0,C 180,E1 -14717.028,E2 -14717.028} C_VEL
LIN {X 0,Y 326.613,Z 71.798,A -85,B 0,C 180,E1 -14720.773,E2 -14720.773} C_VEL
LIN {X 0,Y 326.615,Z 71.797,A -85,B 0,C 180,E1 -14724.481,E2 -14724.481} C_VEL
LIN {X 0,Y 326.61,Z 71.8,A -85,B 0,C 180,E1 -14727.456,E2 -14727.456} C_VEL
LIN {X 0,Y 326.651,Z 71.793,A -85,B 0,C 180,E1 -14730.34,E2 -14730.34} C_VEL
LIN {X 0,Y 326.693,Z 71.791,A -85,B 0,C 180,E1 -14734.517,E2 -14734.517} C_VEL
LIN {X 0,Y 326.652,Z 71.798,A -85,B 0,C 180,E1 -14738.546,E2 -14738.546} C_VEL
LIN {X 0,Y 326.748,Z 71.78,A -85,B 0,C 180,E1 -14741.178,E2 -14741.178} C_VEL
LIN {X 0,Y 326.767,Z 71.776,A -85,B 0,C 180,E1 -14745.433,E2 -14745.433} C_VEL
LIN {X 0,Y 326.763,Z 71.78,A -85,B 0,C 180,E1 -14748.839,E2 -14748.839} C_VEL
LIN {X 0,Y 326.958,Z 71.755,A -85,B 0,C 180,E1 -14752.59,E2 -14752.59} C_VEL
LIN {X 0,Y 326.991,Z 71.752,A -85,B 0,C 180,E1 -14753.831,E2 -14753.831} C_VEL
LIN {X 0,Y 327.047,Z 71.743,A -85,B 0,C 180,E1 -14757.537,E2 -14757.537} C_VEL
LIN {X 0,Y 327.202,Z 71.729,A -85,B 0,C 180,E1 -14760,E2 -14760} C_VEL
LIN {X 0,Y 327.049,Z 71.744,A -85,B 0,C 180,E1 -14762.463,E2 -14762.463} C_VEL
LIN {X 0,Y 326.95,Z 71.757,A -85,B 0,C 180,E1 -14766.17,E2 -14766.17} C_VEL
LIN {X 0,Y 326.787,Z 71.777,A -85,B 0,C 180,E1 -14769.907,E2 -14769.907} C_VEL
LIN {X 0,Y 326.763,Z 71.781,A -85,B 0,C 180,E1 -14773.685,E2 -14773.685} C_VEL
LIN {X 0,Y 326.669,Z 71.794,A -85,B 0,C 180,E1 -14777.53,E2 -14777.53} C_VEL
LIN {X 0,Y 326.657,Z 71.792,A -85,B 0,C 180,E1 -14780.136,E2 -14780.136} C_VEL
LIN {X 0,Y 326.623,Z 71.8,A -85,B 0,C 180,E1 -14782.787,E2 -14782.787} C_VEL
LIN {X 0,Y 326.647,Z 71.795,A -85,B 0,C 180,E1 -14785.488,E2 -14785.488} C_VEL
LIN {X 0,Y 326.631,Z 71.797,A -85,B 0,C 180,E1 -14788.253,E2 -14788.253} C_VEL
LIN {X 0,Y 326.578,Z 71.805,A -85,B 0,C 180,E1 -14791.097,E2 -14791.097} C_VEL
LIN {X 0,Y 326.61,Z 71.799,A -85,B 0,C 180,E1 -14794.019,E2 -14794.019} C_VEL
LIN {X 0,Y 326.631,Z 71.796,A -85,B 0,C 180,E1 -14797.238,E2 -14797.238} C_VEL
LIN {X 0,Y 326.581,Z 71.802,A -85,B 0,C 180,E1 -14801.131,E2 -14801.131} C_VEL
LIN {X 0,Y 326.531,Z 71.81,A -85,B 0,C 180,E1 -14804.743,E2 -14804.743} C_VEL
LIN {X 0,Y 326.577,Z 71.808,A -85,B 0,C 180,E1 -14808.154,E2 -14808.154} C_VEL
LIN {X 0,Y 326.589,Z 71.802,A -85,B 0,C 180,E1 -14811.386,E2 -14811.386} C_VEL
LIN {X 0,Y 326.622,Z 71.798,A -85,B 0,C 180,E1 -14814.851,E2 -14814.851} C_VEL
LIN {X 0,Y 326.661,Z 71.938,A -85,B 0,C 180,E1 -14818.596,E2 -14818.596} C_VEL
LIN {X 0,Y 329.419,Z 84.856,A -85,B 0,C 180,E1 -14822.007,E2 -14822.007} C_VEL
LIN {X 0,Y 330.416,Z 90.61,A -85,B 0,C 180,E1 -14823.469,E2 -14823.469} C_VEL
LIN {X 0,Y 328.961,Z 105.353,A -85,B 0,C 180,E1 -14826.926,E2 -14826.926} C_VEL
LIN {X 0,Y 333.812,Z 143.251,A -85,B 0,C 180,E1 -14828.061,E2 -14828.061} C_VEL
LIN {X 0,Y 334.272,Z 149.363,A -85,B 0,C 180,E1 -14828.222,E2 -14828.222} C_VEL
LIN {X 0,Y 333.12,Z 214.218,A -85,B 0,C 180,E1 -14829.628,E2 -14829.628} C_VEL
LIN {X 0,Y 332.422,Z 227.559,A -85,B 0,C 180,E1 -14830.148,E2 -14830.148} C_VEL
LIN {X 0,Y 331.474,Z 240.352,A -85,B 0,C 180,E1 -14830.894,E2 -14830.894} C_VEL
LIN {X 0,Y 330.392,Z 252.512,A -85,B 0,C 180,E1 -14831.874,E2 -14831.874} C_VEL
LIN {X 0,Y 329.13,Z 264.091,A -85,B 0,C 180,E1 -14833.086,E2 -14833.086} C_VEL
LIN {X 0,Y 328.103,Z 274.784,A -85,B 0,C 180,E1 -14834.504,E2 -14834.504} C_VEL
LIN {X 0,Y 327.171,Z 283.926,A -85,B 0,C 180,E1 -14836.015,E2 -14836.015} C_VEL
LIN {X 0,Y 326.245,Z 293.014,A -85,B 0,C 180,E1 -14837.875,E2 -14837.875} C_VEL
LIN {X 0,Y 325.564,Z 300.325,A -85,B 0,C 180,E1 -14839.741,E2 -14839.741} C_VEL
LIN {X 0,Y 325.267,Z 305.259,A -85,B 0,C 180,E1 -14841.301,E2 -14841.301} C_VEL
LIN {X 0,Y 324.989,Z 310.037,A -85,B 0,C 180,E1 -14843.169,E2 -14843.169} C_VEL
LIN {X 0,Y 324.99,Z 313.687,A -85,B 0,C 180,E1 -14845.038,E2 -14845.038} C_VEL
LIN {X 0,Y 325.016,Z 315.559,A -85,B 0,C 180,E1 -14846.28,E2 -14846.28} C_VEL
LIN {X 0,Y 325.032,Z 316.954,A -85,B 0,C 180,E1 -14847.521,E2 -14847.521} C_VEL
LIN {X 0,Y 325.138,Z 317.946,A -85,B 0,C 180,E1 -14848.761,E2 -14848.761} C_VEL
LIN {X 0,Y 325.191,Z 318.539,A -85,B 0,C 180,E1 -14850,E2 -14850} C_VEL
LIN {X 0,Y 325.062,Z 318.722,A -85,B 0,C 180,E1 -14851.239,E2 -14851.239} C_VEL
LIN {X 0,Y 324.957,Z 317.833,A -85,B 0,C 180,E1 -14853.72,E2 -14853.72} C_VEL
LIN {X 0,Y 324.955,Z 315.377,A -85,B 0,C 180,E1 -14856.208,E2 -14856.208} C_VEL
LIN {X 0,Y 325.184,Z 312.404,A -85,B 0,C 180,E1 -14858.076,E2 -14858.076} C_VEL
LIN {X 0,Y 325.601,Z 308.409,A -85,B 0,C 180,E1 -14859.943,E2 -14859.943} C_VEL
LIN {X 0,Y 326.452,Z 302.315,A -85,B 0,C 180,E1 -14862.117,E2 -14862.117} C_VEL
LIN {X 0,Y 327.737,Z 295.677,A -85,B 0,C 180,E1 -14863.96,E2 -14863.96} C_VEL
LIN {X 0,Y 328.985,Z 288.012,A -85,B 0,C 180,E1 -14865.688,E2 -14865.688} C_VEL
LIN {X 0,Y 330.45,Z 279.096,A -85,B 0,C 180,E1 -14867.323,E2 -14867.323} C_VEL
LIN {X 0,Y 332.242,Z 268.83,A -85,B 0,C 180,E1 -14868.82,E2 -14868.82} C_VEL
LIN {X 0,Y 334.076,Z 257.275,A -85,B 0,C 180,E1 -14870.15,E2 -14870.15} C_VEL
LIN {X 0,Y 335.652,Z 245.9,A -85,B 0,C 180,E1 -14871.173,E2 -14871.173} C_VEL
LIN {X 0,Y 337.02,Z 234.2,A -85,B 0,C 180,E1 -14871.966,E2 -14871.966} C_VEL
LIN {X 0,Y 338.182,Z 220.762,A -85,B 0,C 180,E1 -14872.61,E2 -14872.61} C_VEL
LIN {X 0,Y 338.875,Z 207.438,A -85,B 0,C 180,E1 -14873.005,E2 -14873.005} C_VEL
LIN {X 0,Y 340.221,Z 148.859,A -85,B 0,C 180,E1 -14874.257,E2 -14874.257} C_VEL
LIN {X 0,Y 336.411,Z 125.69,A -85,B 0,C 180,E1 -14875.146,E2 -14875.146} C_VEL
LIN {X 0,Y 332.09,Z 104.395,A -85,B 0,C 180,E1 -14876.098,E2 -14876.098} C_VEL
LIN {X 0,Y 332.767,Z 98.676,A -85,B 0,C 180,E1 -14877.496,E2 -14877.496} C_VEL
LIN {X 0,Y 331.292,Z 91.219,A -85,B 0,C 180,E1 -14879.568,E2 -14879.568} C_VEL
LIN {X 0,Y 328.875,Z 80.591,A -85,B 0,C 180,E1 -14882.674,E2 -14882.674} C_VEL
LIN {X 0,Y 326.666,Z 71.794,A -85,B 0,C 180,E1 -14885.454,E2 -14885.454} C_VEL
LIN {X 0,Y 326.613,Z 71.787,A -85,B 0,C 180,E1 -14889.227,E2 -14889.227} C_VEL
LIN {X 0,Y 326.578,Z 71.801,A -85,B 0,C 180,E1 -14892.972,E2 -14892.972} C_VEL
LIN {X 0,Y 326.578,Z 71.798,A -85,B 0,C 180,E1 -14897.028,E2 -14897.028} C_VEL
LIN {X 0,Y 326.614,Z 71.792,A -85,B 0,C 180,E1 -14900.773,E2 -14900.773} C_VEL
LIN {X 0,Y 326.615,Z 71.796,A -85,B 0,C 180,E1 -14904.48,E2 -14904.48} C_VEL
LIN {X 0,Y 326.61,Z 71.799,A -85,B 0,C 180,E1 -14907.456,E2 -14907.456} C_VEL
LIN {X 0,Y 326.663,Z 71.787,A -85,B 0,C 180,E1 -14910.341,E2 -14910.341} C_VEL
LIN {X 0,Y 326.693,Z 71.783,A -85,B 0,C 180,E1 -14914.516,E2 -14914.516} C_VEL
LIN {X 0,Y 326.649,Z 71.788,A -85,B 0,C 180,E1 -14918.545,E2 -14918.545} C_VEL
LIN {X 0,Y 326.747,Z 71.782,A -85,B 0,C 180,E1 -14921.177,E2 -14921.177} C_VEL
LIN {X 0,Y 326.766,Z 71.78,A -85,B 0,C 180,E1 -14925.433,E2 -14925.433} C_VEL
LIN {X 0,Y 326.773,Z 71.776,A -85,B 0,C 180,E1 -14928.839,E2 -14928.839} C_VEL
LIN {X 0,Y 326.961,Z 71.745,A -85,B 0,C 180,E1 -14932.59,E2 -14932.59} C_VEL
LIN {X 0,Y 326.992,Z 71.743,A -85,B 0,C 180,E1 -14933.831,E2 -14933.831} C_VEL
LIN {X 0,Y 327.046,Z 71.74,A -85,B 0,C 180,E1 -14937.537,E2 -14937.537} C_VEL
LIN {X 0,Y 327.201,Z 71.725,A -85,B 0,C 180,E1 -14940,E2 -14940} C_VEL
LIN {X 0,Y 327.048,Z 71.741,A -85,B 0,C 180,E1 -14942.463,E2 -14942.463} C_VEL
LIN {X 0,Y 326.954,Z 71.755,A -85,B 0,C 180,E1 -14946.586,E2 -14946.586} C_VEL
LIN {X 0,Y 326.786,Z 71.774,A -85,B 0,C 180,E1 -14949.907,E2 -14949.907} C_VEL
LIN {X 0,Y 326.762,Z 71.772,A -85,B 0,C 180,E1 -14953.685,E2 -14953.685} C_VEL
LIN {X 0,Y 326.667,Z 71.789,A -85,B 0,C 180,E1 -14957.53,E2 -14957.53} C_VEL
LIN {X 0,Y 326.66,Z 71.792,A -85,B 0,C 180,E1 -14960.135,E2 -14960.135} C_VEL
LIN {X 0,Y 326.649,Z 71.792,A -85,B 0,C 180,E1 -14964.129,E2 -14964.129} C_VEL
LIN {X 0,Y 326.629,Z 71.796,A -85,B 0,C 180,E1 -14968.253,E2 -14968.253} C_VEL
LIN {X 0,Y 326.576,Z 71.801,A -85,B 0,C 180,E1 -14971.097,E2 -14971.097} C_VEL
LIN {X 0,Y 326.608,Z 71.797,A -85,B 0,C 180,E1 -14974.019,E2 -14974.019} C_VEL
LIN {X 0,Y 326.624,Z 71.796,A -85,B 0,C 180,E1 -14977.237,E2 -14977.237} C_VEL
LIN {X 0,Y 326.575,Z 71.79,A -85,B 0,C 180,E1 -14981.13,E2 -14981.13} C_VEL
LIN {X 0,Y 326.528,Z 71.813,A -85,B 0,C 180,E1 -14984.743,E2 -14984.743} C_VEL
LIN {X 0,Y 326.576,Z 71.806,A -85,B 0,C 180,E1 -14988.154,E2 -14988.154} C_VEL
LIN {X 0,Y 326.589,Z 71.805,A -85,B 0,C 180,E1 -14992.131,E2 -14992.131} C_VEL
LIN {X 0,Y 326.612,Z 71.835,A -85,B 0,C 180,E1 -14992.642,E2 -14992.642} C_VEL
LIN {X 0,Y 327.155,Z 74.143,A -85,B 0,C 180,E1 -14993.458,E2 -14993.458} C_VEL
LIN {X 0,Y 336.337,Z 93.182,A -85,B 0,C 180,E1 -14994.856,E2 -14994.856} C_VEL
LIN {X 0,Y 341.282,Z 104.993,A -85,B 0,C 180,E1 -14995.595,E2 -14995.595} C_VEL
LIN {X 0,Y 339.249,Z 181.015,A -85,B 0,C 180,E1 -14997.236,E2 -14997.236} C_VEL
LIN {X 0,Y 338.571,Z 194.392,A -85,B 0,C 180,E1 -14997.777,E2 -14997.777} C_VEL
LIN {X 0,Y 337.738,Z 207.173,A -85,B 0,C 180,E1 -14998.558,E2 -14998.558} C_VEL
LIN {X 0,Y 336.602,Z 217.784,A -85,B 0,C 180,E1 -14999.411,E2 -14999.411} C_VEL
LIN {X 0,Y 335.04,Z 229.607,A -85,B 0,C 180,E1 -15000.638,E2 -15000.638} C_VEL
LIN {X 0,Y 333.475,Z 240.217,A -85,B 0,C 180,E1 -15002.036,E2 -15002.036} C_VEL
LIN {X 0,Y 331.834,Z 249.65,A -85,B 0,C 180,E1 -15003.592,E2 -15003.592} C_VEL
LIN {X 0,Y 330.197,Z 258.741,A -85,B 0,C 180,E1 -15005.478,E2 -15005.478} C_VEL
LIN {X 0,Y 328.807,Z 265.99,A -85,B 0,C 180,E1 -15007.373,E2 -15007.373} C_VEL
LIN {X 0,Y 327.63,Z 271.703,A -85,B 0,C 180,E1 -15009.271,E2 -15009.271} C_VEL
LIN {X 0,Y 326.791,Z 276.158,A -85,B 0,C 180,E1 -15011.18,E2 -15011.18} C_VEL
LIN {X 0,Y 326.295,Z 278.493,A -85,B 0,C 180,E1 -15012.45,E2 -15012.45} C_VEL
LIN {X 0,Y 325.894,Z 280.385,A -85,B 0,C 180,E1 -15013.719,E2 -15013.719} C_VEL
LIN {X 0,Y 325.55,Z 281.802,A -85,B 0,C 180,E1 -15014.986,E2 -15014.986} C_VEL
LIN {X 0,Y 325.338,Z 282.9,A -85,B 0,C 180,E1 -15016.433,E2 -15016.433} C_VEL
LIN {X 0,Y 325.044,Z 283.585,A -85,B 0,C 180,E1 -15018.779,E2 -15018.779} C_VEL
LIN {X 0,Y 324.994,Z 283.345,A -85,B 0,C 180,E1 -15020.038,E2 -15020.038} C_VEL
LIN {X 0,Y 325.126,Z 281.688,A -85,B 0,C 180,E1 -15022.548,E2 -15022.548} C_VEL
LIN {X 0,Y 325.3,Z 280.255,A -85,B 0,C 180,E1 -15023.799,E2 -15023.799} C_VEL
LIN {X 0,Y 325.41,Z 277.306,A -85,B 0,C 180,E1 -15025.665,E2 -15025.665} C_VEL
LIN {X 0,Y 325.807,Z 273.309,A -85,B 0,C 180,E1 -15027.527,E2 -15027.527} C_VEL
LIN {X 0,Y 326.329,Z 267.18,A -85,B 0,C 180,E1 -15029.692,E2 -15029.692} C_VEL
LIN {X 0,Y 327.143,Z 260.489,A -85,B 0,C 180,E1 -15031.539,E2 -15031.539} C_VEL
LIN {X 0,Y 327.987,Z 252.219,A -85,B 0,C 180,E1 -15033.378,E2 -15033.378} C_VEL
LIN {X 0,Y 328.834,Z 243.71,A -85,B 0,C 180,E1 -15034.904,E2 -15034.904} C_VEL
LIN {X 0,Y 330.035,Z 234.331,A -85,B 0,C 180,E1 -15036.266,E2 -15036.266} C_VEL
LIN {X 0,Y 331.159,Z 222.746,A -85,B 0,C 180,E1 -15037.622,E2 -15037.622} C_VEL
LIN {X 0,Y 332.072,Z 211.263,A -85,B 0,C 180,E1 -15038.673,E2 -15038.673} C_VEL
LIN {X 0,Y 332.771,Z 199.381,A -85,B 0,C 180,E1 -15039.497,E2 -15039.497} C_VEL
LIN {X 0,Y 333.327,Z 186.528,A -85,B 0,C 180,E1 -15040.133,E2 -15040.133} C_VEL
LIN {X 0,Y 333.71,Z 174.453,A -85,B 0,C 180,E1 -15040.504,E2 -15040.504} C_VEL
LIN {X 0,Y 335.053,Z 96.983,A -85,B 0,C 180,E1 -15042.154,E2 -15042.154} C_VEL
LIN {X 0,Y 327.594,Z 74.923,A -85,B 0,C 180,E1 -15043.109,E2 -15043.109} C_VEL
LIN {X 0,Y 327.017,Z 73.132,A -85,B 0,C 180,E1 -15043.195,E2 -15043.195} C_VEL
LIN {X 0,Y 326.76,Z 71.783,A -85,B 0,C 180,E1 -15043.686,E2 -15043.686} C_VEL
LIN {X 0,Y 326.701,Z 71.787,A -85,B 0,C 180,E1 -15047.528,E2 -15047.528} C_VEL
LIN {X 0,Y 326.662,Z 71.795,A -85,B 0,C 180,E1 -15050.135,E2 -15050.135} C_VEL
LIN {X 0,Y 326.65,Z 71.798,A -85,B 0,C 180,E1 -15054.129,E2 -15054.129} C_VEL
LIN {X 0,Y 326.673,Z 71.79,A -85,B 0,C 180,E1 -15057.008,E2 -15057.008} C_VEL
LIN {X 0,Y 326.635,Z 71.796,A -85,B 0,C 180,E1 -15060.61,E2 -15060.61} C_VEL
LIN {X 0,Y 326.598,Z 71.799,A -85,B 0,C 180,E1 -15062.373,E2 -15062.373} C_VEL
LIN {X 0,Y 325.987,Z 71.882,A -85,B 0,C 180,E1 -15063.402,E2 -15063.402} C_VEL
LIN {X 0,Y 323.152,Z 72.24,A -85,B 0,C 180,E1 -15065.078,E2 -15065.078} C_VEL
LIN {X 0,Y 320.714,Z 72.541,A -85,B 0,C 180,E1 -15066.435,E2 -15066.435} C_VEL
LIN {X 0,Y 319.662,Z 72.669,A -85,B 0,C 180,E1 -15067.486,E2 -15067.486} C_VEL
LIN {X 0,Y 319.576,Z 72.678,A -85,B 0,C 180,E1 -15067.843,E2 -15067.843} C_VEL
LIN {X 0,Y 319.553,Z 72.682,A -85,B 0,C 180,E1 -15071.603,E2 -15071.603} C_VEL
LIN {X 0,Y 319.49,Z 72.688,A -85,B 0,C 180,E1 -15075.258,E2 -15075.258} C_VEL
LIN {X 0,Y 319.53,Z 72.68,A -85,B 0,C 180,E1 -15078.712,E2 -15078.712} C_VEL
LIN {X 0,Y 319.564,Z 72.676,A -85,B 0,C 180,E1 -15082.348,E2 -15082.348} C_VEL
LIN {X 0,Y 319.563,Z 72.68,A -85,B 0,C 180,E1 -15085.124,E2 -15085.124} C_VEL
LIN {X 0,Y 319.569,Z 72.679,A -85,B 0,C 180,E1 -15089.059,E2 -15089.059} C_VEL
LIN {X 0,Y 319.609,Z 72.673,A -85,B 0,C 180,E1 -15092.498,E2 -15092.498} C_VEL
LIN {X 0,Y 319.608,Z 72.671,A -85,B 0,C 180,E1 -15095.304,E2 -15095.304} C_VEL
LIN {X 0,Y 319.601,Z 72.672,A -85,B 0,C 180,E1 -15098.048,E2 -15098.048} C_VEL
LIN {X 0,Y 319.692,Z 72.659,A -85,B 0,C 180,E1 -15100.963,E2 -15100.963} C_VEL
LIN {X 0,Y 319.735,Z 72.652,A -85,B 0,C 180,E1 -15105.276,E2 -15105.276} C_VEL
LIN {X 0,Y 319.719,Z 72.659,A -85,B 0,C 180,E1 -15108.59,E2 -15108.59} C_VEL
LIN {X 0,Y 319.912,Z 72.633,A -85,B 0,C 180,E1 -15112.426,E2 -15112.426} C_VEL
LIN {X 0,Y 319.744,Z 72.648,A -85,B 0,C 180,E1 -15114.956,E2 -15114.956} C_VEL
LIN {X 0,Y 319.991,Z 72.621,A -85,B 0,C 180,E1 -15117.483,E2 -15117.483} C_VEL
LIN {X 0,Y 320.154,Z 72.607,A -85,B 0,C 180,E1 -15120,E2 -15120} C_VEL
LIN {X 0,Y 319.993,Z 72.623,A -85,B 0,C 180,E1 -15122.518,E2 -15122.518} C_VEL
LIN {X 0,Y 319.907,Z 72.634,A -85,B 0,C 180,E1 -15126.307,E2 -15126.307} C_VEL
LIN {X 0,Y 319.74,Z 72.654,A -85,B 0,C 180,E1 -15130.128,E2 -15130.128} C_VEL
LIN {X 0,Y 319.736,Z 72.655,A -85,B 0,C 180,E1 -15133.992,E2 -15133.992} C_VEL
LIN {X 0,Y 319.629,Z 72.668,A -85,B 0,C 180,E1 -15137.929,E2 -15137.929} C_VEL
LIN {X 0,Y 319.612,Z 72.671,A -85,B 0,C 180,E1 -15140.599,E2 -15140.599} C_VEL
LIN {X 0,Y 319.571,Z 72.678,A -85,B 0,C 180,E1 -15143.32,E2 -15143.32} C_VEL
LIN {X 0,Y 319.583,Z 72.674,A -85,B 0,C 180,E1 -15146.093,E2 -15146.093} C_VEL
LIN {X 0,Y 319.561,Z 72.681,A -85,B 0,C 180,E1 -15148.937,E2 -15148.937} C_VEL
LIN {X 0,Y 319.528,Z 72.681,A -85,B 0,C 180,E1 -15151.862,E2 -15151.862} C_VEL
LIN {X 0,Y 319.583,Z 72.674,A -85,B 0,C 180,E1 -15155.543,E2 -15155.543} C_VEL
LIN {X 0,Y 319.56,Z 72.678,A -85,B 0,C 180,E1 -15158.01,E2 -15158.01} C_VEL
LIN {X 0,Y 319.529,Z 72.681,A -85,B 0,C 180,E1 -15161.597,E2 -15161.597} C_VEL
LIN {X 0,Y 319.491,Z 72.685,A -85,B 0,C 180,E1 -15165.257,E2 -15165.257} C_VEL
LIN {X 0,Y 319.528,Z 72.682,A -85,B 0,C 180,E1 -15168.711,E2 -15168.711} C_VEL
LIN {X 0,Y 319.551,Z 72.68,A -85,B 0,C 180,E1 -15172.351,E2 -15172.351} C_VEL
LIN {X 0,Y 319.562,Z 72.678,A -85,B 0,C 180,E1 -15175.123,E2 -15175.123} C_VEL
LIN {X 0,Y 319.608,Z 72.86,A -85,B 0,C 180,E1 -15178.27,E2 -15178.27} C_VEL
LIN {X 0,Y 322.348,Z 85.484,A -85,B 0,C 180,E1 -15181.692,E2 -15181.692} C_VEL
LIN {X 0,Y 323.413,Z 91.351,A -85,B 0,C 180,E1 -15183.222,E2 -15183.222} C_VEL
LIN {X 0,Y 322.549,Z 100.996,A -85,B 0,C 180,E1 -15185.544,E2 -15185.544} C_VEL
LIN {X 0,Y 322.106,Z 104.932,A -85,B 0,C 180,E1 -15186.482,E2 -15186.482} C_VEL
LIN {X 0,Y 326.904,Z 142.41,A -85,B 0,C 180,E1 -15187.647,E2 -15187.647} C_VEL
LIN {X 0,Y 327.538,Z 149.52,A -85,B 0,C 180,E1 -15187.846,E2 -15187.846} C_VEL
LIN {X 0,Y 326.335,Z 213.874,A -85,B 0,C 180,E1 -15189.268,E2 -15189.268} C_VEL
LIN {X 0,Y 325.61,Z 227.204,A -85,B 0,C 180,E1 -15189.797,E2 -15189.797} C_VEL
LIN {X 0,Y 324.659,Z 239.998,A -85,B 0,C 180,E1 -15190.559,E2 -15190.559} C_VEL
LIN {X 0,Y 323.559,Z 251.343,A -85,B 0,C 180,E1 -15191.478,E2 -15191.478} C_VEL
LIN {X 0,Y 322.281,Z 263.073,A -85,B 0,C 180,E1 -15192.715,E2 -15192.715} C_VEL
LIN {X 0,Y 321.226,Z 273.65,A -85,B 0,C 180,E1 -15194.129,E2 -15194.129} C_VEL
LIN {X 0,Y 320.255,Z 283.146,A -85,B 0,C 180,E1 -15195.707,E2 -15195.707} C_VEL
LIN {X 0,Y 319.402,Z 290.924,A -85,B 0,C 180,E1 -15197.289,E2 -15197.289} C_VEL
LIN {X 0,Y 318.594,Z 298.531,A -85,B 0,C 180,E1 -15199.193,E2 -15199.193} C_VEL
LIN {X 0,Y 318.191,Z 304.651,A -85,B 0,C 180,E1 -15201.106,E2 -15201.106} C_VEL
LIN {X 0,Y 317.914,Z 309.479,A -85,B 0,C 180,E1 -15203.016,E2 -15203.016} C_VEL
LIN {X 0,Y 317.894,Z 313.172,A -85,B 0,C 180,E1 -15204.926,E2 -15204.926} C_VEL
LIN {X 0,Y 317.94,Z 315.075,A -85,B 0,C 180,E1 -15206.198,E2 -15206.198} C_VEL
LIN {X 0,Y 317.942,Z 316.501,A -85,B 0,C 180,E1 -15207.466,E2 -15207.466} C_VEL
LIN {X 0,Y 318.043,Z 317.513,A -85,B 0,C 180,E1 -15208.734,E2 -15208.734} C_VEL
LIN {X 0,Y 318.114,Z 318.126,A -85,B 0,C 180,E1 -15210,E2 -15210} C_VEL
LIN {X 0,Y 317.966,Z 318.334,A -85,B 0,C 180,E1 -15211.266,E2 -15211.266} C_VEL
LIN {X 0,Y 317.868,Z 318.114,A -85,B 0,C 180,E1 -15212.534,E2 -15212.534} C_VEL
LIN {X 0,Y 317.88,Z 317.495,A -85,B 0,C 180,E1 -15213.803,E2 -15213.803} C_VEL
LIN {X 0,Y 317.882,Z 315.081,A -85,B 0,C 180,E1 -15216.347,E2 -15216.347} C_VEL
LIN {X 0,Y 318.142,Z 312.145,A -85,B 0,C 180,E1 -15218.256,E2 -15218.256} C_VEL
LIN {X 0,Y 318.569,Z 308.193,A -85,B 0,C 180,E1 -15220.165,E2 -15220.165} C_VEL
LIN {X 0,Y 319.315,Z 303.133,A -85,B 0,C 180,E1 -15222.069,E2 -15222.069} C_VEL
LIN {X 0,Y 320.595,Z 296.815,A -85,B 0,C 180,E1 -15223.954,E2 -15223.954} C_VEL
LIN {X 0,Y 321.887,Z 289.408,A -85,B 0,C 180,E1 -15225.735,E2 -15225.735} C_VEL
LIN {X 0,Y 323.377,Z 280.94,A -85,B 0,C 180,E1 -15227.387,E2 -15227.387} C_VEL
LIN {X 0,Y 325.146,Z 271.21,A -85,B 0,C 180,E1 -15228.919,E2 -15228.919} C_VEL
LIN {X 0,Y 326.994,Z 260.42,A -85,B 0,C 180,E1 -15230.278,E2 -15230.278} C_VEL
LIN {X 0,Y 328.599,Z 249.921,A -85,B 0,C 180,E1 -15231.321,E2 -15231.321} C_VEL
LIN {X 0,Y 330.109,Z 238.434,A -85,B 0,C 180,E1 -15232.204,E2 -15232.204} C_VEL
LIN {X 0,Y 331.44,Z 225.502,A -85,B 0,C 180,E1 -15232.932,E2 -15232.932} C_VEL
LIN {X 0,Y 332.253,Z 212.989,A -85,B 0,C 180,E1 -15233.408,E2 -15233.408} C_VEL
LIN {X 0,Y 333.916,Z 149.854,A -85,B 0,C 180,E1 -15234.797,E2 -15234.797} C_VEL
LIN {X 0,Y 330.153,Z 126.74,A -85,B 0,C 180,E1 -15235.708,E2 -15235.708} C_VEL
LIN {X 0,Y 325.481,Z 104.082,A -85,B 0,C 180,E1 -15236.737,E2 -15236.737} C_VEL
LIN {X 0,Y 325.865,Z 99.732,A -85,B 0,C 180,E1 -15237.839,E2 -15237.839} C_VEL
LIN {X 0,Y 323.788,Z 89.93,A -85,B 0,C 180,E1 -15240.669,E2 -15240.669} C_VEL
LIN {X 0,Y 321.354,Z 79.697,A -85,B 0,C 180,E1 -15243.792,E2 -15243.792} C_VEL
LIN {X 0,Y 319.593,Z 72.677,A -85,B 0,C 180,E1 -15246.053,E2 -15246.053} C_VEL
LIN {X 0,Y 319.56,Z 72.665,A -85,B 0,C 180,E1 -15249.669,E2 -15249.669} C_VEL
LIN {X 0,Y 319.524,Z 72.682,A -85,B 0,C 180,E1 -15253.461,E2 -15253.461} C_VEL
LIN {X 0,Y 319.556,Z 72.672,A -85,B 0,C 180,E1 -15257.017,E2 -15257.017} C_VEL
LIN {X 0,Y 319.549,Z 72.671,A -85,B 0,C 180,E1 -15260.371,E2 -15260.371} C_VEL
LIN {X 0,Y 319.561,Z 72.672,A -85,B 0,C 180,E1 -15263.572,E2 -15263.572} C_VEL
LIN {X 0,Y 319.579,Z 72.669,A -85,B 0,C 180,E1 -15266.686,E2 -15266.686} C_VEL
LIN {X 0,Y 319.594,Z 72.668,A -85,B 0,C 180,E1 -15269.617,E2 -15269.617} C_VEL
LIN {X 0,Y 319.612,Z 72.674,A -85,B 0,C 180,E1 -15272.498,E2 -15272.498} C_VEL
LIN {X 0,Y 319.609,Z 72.673,A -85,B 0,C 180,E1 -15275.304,E2 -15275.304} C_VEL
LIN {X 0,Y 319.6,Z 72.666,A -85,B 0,C 180,E1 -15278.048,E2 -15278.048} C_VEL
LIN {X 0,Y 319.692,Z 72.662,A -85,B 0,C 180,E1 -15280.962,E2 -15280.962} C_VEL
LIN {X 0,Y 319.734,Z 72.656,A -85,B 0,C 180,E1 -15285.276,E2 -15285.276} C_VEL
LIN {X 0,Y 319.756,Z 72.653,A -85,B 0,C 180,E1 -15289.873,E2 -15289.873} C_VEL
LIN {X 0,Y 319.916,Z 72.624,A -85,B 0,C 180,E1 -15292.426,E2 -15292.426} C_VEL
LIN {X 0,Y 319.745,Z 72.654,A -85,B 0,C 180,E1 -15294.956,E2 -15294.956} C_VEL
LIN {X 0,Y 319.99,Z 72.619,A -85,B 0,C 180,E1 -15297.482,E2 -15297.482} C_VEL
LIN {X 0,Y 320.152,Z 72.603,A -85,B 0,C 180,E1 -15300,E2 -15300} C_VEL
LIN {X 0,Y 319.992,Z 72.619,A -85,B 0,C 180,E1 -15302.517,E2 -15302.517} C_VEL
LIN {X 0,Y 319.916,Z 72.632,A -85,B 0,C 180,E1 -15306.571,E2 -15306.571} C_VEL
LIN {X 0,Y 319.738,Z 72.654,A -85,B 0,C 180,E1 -15310.128,E2 -15310.128} C_VEL
LIN {X 0,Y 319.735,Z 72.646,A -85,B 0,C 180,E1 -15313.992,E2 -15313.992} C_VEL
LIN {X 0,Y 319.627,Z 72.664,A -85,B 0,C 180,E1 -15317.929,E2 -15317.929} C_VEL
LIN {X 0,Y 319.614,Z 72.672,A -85,B 0,C 180,E1 -15320.599,E2 -15320.599} C_VEL
LIN {X 0,Y 319.57,Z 72.671,A -85,B 0,C 180,E1 -15323.319,E2 -15323.319} C_VEL
LIN {X 0,Y 319.581,Z 72.676,A -85,B 0,C 180,E1 -15326.093,E2 -15326.093} C_VEL
LIN {X 0,Y 319.56,Z 72.68,A -85,B 0,C 180,E1 -15328.936,E2 -15328.936} C_VEL
LIN {X 0,Y 319.526,Z 72.682,A -85,B 0,C 180,E1 -15331.862,E2 -15331.862} C_VEL
LIN {X 0,Y 319.581,Z 72.677,A -85,B 0,C 180,E1 -15335.543,E2 -15335.543} C_VEL
LIN {X 0,Y 319.56,Z 72.672,A -85,B 0,C 180,E1 -15339.668,E2 -15339.668} C_VEL
LIN {X 0,Y 319.522,Z 72.687,A -85,B 0,C 180,E1 -15343.46,E2 -15343.46} C_VEL
LIN {X 0,Y 319.555,Z 72.682,A -85,B 0,C 180,E1 -15347.016,E2 -15347.016} C_VEL
LIN {X 0,Y 319.545,Z 72.682,A -85,B 0,C 180,E1 -15350.37,E2 -15350.37} C_VEL
LIN {X 0,Y 319.56,Z 72.815,A -85,B 0,C 180,E1 -15352.064,E2 -15352.064} C_VEL
LIN {X 0,Y 320.047,Z 74.699,A -85,B 0,C 180,E1 -15352.733,E2 -15352.733} C_VEL
LIN {X 0,Y 329.443,Z 93.794,A -85,B 0,C 180,E1 -15354.198,E2 -15354.198} C_VEL
LIN {X 0,Y 334.988,Z 106.765,A -85,B 0,C 180,E1 -15355.055,E2 -15355.055} C_VEL
LIN {X 0,Y 332.936,Z 181.041,A -85,B 0,C 180,E1 -15356.683,E2 -15356.683} C_VEL
LIN {X 0,Y 332.24,Z 194.299,A -85,B 0,C 180,E1 -15357.221,E2 -15357.221} C_VEL
LIN {X 0,Y 331.406,Z 206.749,A -85,B 0,C 180,E1 -15357.983,E2 -15357.983} C_VEL
LIN {X 0,Y 330.248,Z 217.199,A -85,B 0,C 180,E1 -15358.817,E2 -15358.817} C_VEL
LIN {X 0,Y 328.675,Z 228.801,A -85,B 0,C 180,E1 -15360.012,E2 -15360.012} C_VEL
LIN {X 0,Y 327.024,Z 239.618,A -85,B 0,C 180,E1 -15361.434,E2 -15361.434} C_VEL
LIN {X 0,Y 325.303,Z 249.286,A -85,B 0,C 180,E1 -15363.019,E2 -15363.019} C_VEL
LIN {X 0,Y 323.565,Z 258.508,A -85,B 0,C 180,E1 -15364.941,E2 -15364.941} C_VEL
LIN {X 0,Y 322.073,Z 265.881,A -85,B 0,C 180,E1 -15366.872,E2 -15366.872} C_VEL
LIN {X 0,Y 320.822,Z 271.721,A -85,B 0,C 180,E1 -15368.81,E2 -15368.81} C_VEL
LIN {X 0,Y 319.829,Z 276.516,A -85,B 0,C 180,E1 -15370.89,E2 -15370.89} C_VEL
LIN {X 0,Y 318.912,Z 280.569,A -85,B 0,C 180,E1 -15373.352,E2 -15373.352} C_VEL
LIN {X 0,Y 318.543,Z 282.061,A -85,B 0,C 180,E1 -15374.648,E2 -15374.648} C_VEL
LIN {X 0,Y 318.28,Z 283.304,A -85,B 0,C 180,E1 -15376.305,E2 -15376.305} C_VEL
LIN {X 0,Y 317.97,Z 283.962,A -85,B 0,C 180,E1 -15378.526,E2 -15378.526} C_VEL
LIN {X 0,Y 317.904,Z 283.789,A -85,B 0,C 180,E1 -15379.813,E2 -15379.813} C_VEL
LIN {X 0,Y 317.938,Z 283.189,A -85,B 0,C 180,E1 -15381.099,E2 -15381.099} C_VEL
LIN {X 0,Y 318.226,Z 280.822,A -85,B 0,C 180,E1 -15383.66,E2 -15383.66} C_VEL
LIN {X 0,Y 318.326,Z 277.939,A -85,B 0,C 180,E1 -15385.568,E2 -15385.568} C_VEL
LIN {X 0,Y 318.72,Z 274.024,A -85,B 0,C 180,E1 -15387.472,E2 -15387.472} C_VEL
LIN {X 0,Y 319.134,Z 268.998,A -85,B 0,C 180,E1 -15389.369,E2 -15389.369} C_VEL
LIN {X 0,Y 319.89,Z 262.66,A -85,B 0,C 180,E1 -15391.259,E2 -15391.259} C_VEL
LIN {X 0,Y 320.773,Z 254.754,A -85,B 0,C 180,E1 -15393.14,E2 -15393.14} C_VEL
LIN {X 0,Y 321.8,Z 244.948,A -85,B 0,C 180,E1 -15395.012,E2 -15395.012} C_VEL
LIN {X 0,Y 323.032,Z 235.767,A -85,B 0,C 180,E1 -15396.402,E2 -15396.402} C_VEL
LIN {X 0,Y 324.194,Z 224.402,A -85,B 0,C 180,E1 -15397.787,E2 -15397.787} C_VEL
LIN {X 0,Y 325.15,Z 213.265,A -85,B 0,C 180,E1 -15398.859,E2 -15398.859} C_VEL
LIN {X 0,Y 325.923,Z 200.79,A -85,B 0,C 180,E1 -15399.777,E2 -15399.777} C_VEL
LIN {X 0,Y 326.526,Z 187.45,A -85,B 0,C 180,E1 -15400.463,E2 -15400.463} C_VEL
LIN {X 0,Y 326.964,Z 174.198,A -85,B 0,C 180,E1 -15400.88,E2 -15400.88} C_VEL
LIN {X 0,Y 328.257,Z 97.958,A -85,B 0,C 180,E1 -15402.54,E2 -15402.54} C_VEL
LIN {X 0,Y 320.557,Z 75.513,A -85,B 0,C 180,E1 -15403.551,E2 -15403.551} C_VEL
LIN {X 0,Y 319.857,Z 73.382,A -85,B 0,C 180,E1 -15403.688,E2 -15403.688} C_VEL
LIN {X 0,Y 319.733,Z 72.659,A -85,B 0,C 180,E1 -15403.992,E2 -15403.992} C_VEL
LIN {X 0,Y 319.66,Z 72.666,A -85,B 0,C 180,E1 -15407.927,E2 -15407.927} C_VEL
LIN {X 0,Y 319.605,Z 72.673,A -85,B 0,C 180,E1 -15410.6,E2 -15410.6} C_VEL
LIN {X 0,Y 319.604,Z 72.672,A -85,B 0,C 180,E1 -15414.696,E2 -15414.696} C_VEL
LIN {X 0,Y 319.612,Z 72.673,A -85,B 0,C 180,E1 -15418.41,E2 -15418.41} C_VEL
LIN {X 0,Y 319.533,Z 72.684,A -85,B 0,C 180,E1 -15421.862,E2 -15421.862} C_VEL
LIN {X 0,Y 319.582,Z 72.677,A -85,B 0,C 180,E1 -15425.544,E2 -15425.544} C_VEL
LIN {X 0,Y 319.576,Z 72.678,A -85,B 0,C 180,E1 -15427.843,E2 -15427.843} C_VEL
LIN {X 0,Y 318.902,Z 72.76,A -85,B 0,C 180,E1 -15428.894,E2 -15428.894} C_VEL
LIN {X 0,Y 316.027,Z 73.116,A -85,B 0,C 180,E1 -15430.604,E2 -15430.604} C_VEL
LIN {X 0,Y 313.588,Z 73.422,A -85,B 0,C 180,E1 -15431.99,E2 -15431.99} C_VEL
LIN {X 0,Y 312.54,Z 73.552,A -85,B 0,C 180,E1 -15433.063,E2 -15433.063} C_VEL
LIN {X 0,Y 312.453,Z 73.559,A -85,B 0,C 180,E1 -15433.427,E2 -15433.427} C_VEL
LIN {X 0,Y 312.492,Z 73.56,A -85,B 0,C 180,E1 -15437.569,E2 -15437.569} C_VEL
LIN {X 0,Y 312.505,Z 73.557,A -85,B 0,C 180,E1 -15440.972,E2 -15440.972} C_VEL
LIN {X 0,Y 312.534,Z 73.55,A -85,B 0,C 180,E1 -15444.221,E2 -15444.221} C_VEL
LIN {X 0,Y 312.506,Z 73.557,A -85,B 0,C 180,E1 -15447.334,E2 -15447.334} C_VEL
LIN {X 0,Y 312.547,Z 73.552,A -85,B 0,C 180,E1 -15451.279,E2 -15451.279} C_VEL
LIN {X 0,Y 312.589,Z 73.549,A -85,B 0,C 180,E1 -15454.711,E2 -15454.711} C_VEL
LIN {X 0,Y 312.591,Z 73.545,A -85,B 0,C 180,E1 -15457.529,E2 -15457.529} C_VEL
LIN {X 0,Y 312.642,Z 73.535,A -85,B 0,C 180,E1 -15461.657,E2 -15461.657} C_VEL
LIN {X 0,Y 312.698,Z 73.528,A -85,B 0,C 180,E1 -15465.687,E2 -15465.687} C_VEL
LIN {X 0,Y 312.69,Z 73.533,A -85,B 0,C 180,E1 -15469.642,E2 -15469.642} C_VEL
LIN {X 0,Y 312.848,Z 73.514,A -85,B 0,C 180,E1 -15472.254,E2 -15472.254} C_VEL
LIN {X 0,Y 312.902,Z 73.504,A -85,B 0,C 180,E1 -15473.552,E2 -15473.552} C_VEL
LIN {X 0,Y 312.937,Z 73.498,A -85,B 0,C 180,E1 -15477.426,E2 -15477.426} C_VEL
LIN {X 0,Y 313.106,Z 73.484,A -85,B 0,C 180,E1 -15480,E2 -15480} C_VEL
LIN {X 0,Y 312.939,Z 73.501,A -85,B 0,C 180,E1 -15482.575,E2 -15482.575} C_VEL
LIN {X 0,Y 312.85,Z 73.512,A -85,B 0,C 180,E1 -15486.449,E2 -15486.449} C_VEL
LIN {X 0,Y 312.755,Z 73.525,A -85,B 0,C 180,E1 -15489.05,E2 -15489.05} C_VEL
LIN {X 0,Y 312.639,Z 73.541,A -85,B 0,C 180,E1 -15492.991,E2 -15492.991} C_VEL
LIN {X 0,Y 312.626,Z 73.542,A -85,B 0,C 180,E1 -15495.651,E2 -15495.651} C_VEL
LIN {X 0,Y 312.581,Z 73.546,A -85,B 0,C 180,E1 -15499.71,E2 -15499.71} C_VEL
LIN {X 0,Y 312.548,Z 73.553,A -85,B 0,C 180,E1 -15502.789,E2 -15502.789} C_VEL
LIN {X 0,Y 312.541,Z 73.551,A -85,B 0,C 180,E1 -15505.911,E2 -15505.911} C_VEL
LIN {X 0,Y 312.507,Z 73.556,A -85,B 0,C 180,E1 -15509.654,E2 -15509.654} C_VEL
LIN {X 0,Y 312.523,Z 73.554,A -85,B 0,C 180,E1 -15513.689,E2 -15513.689} C_VEL
LIN {X 0,Y 312.529,Z 73.553,A -85,B 0,C 180,E1 -15517.385,E2 -15517.385} C_VEL
LIN {X 0,Y 312.493,Z 73.56,A -85,B 0,C 180,E1 -15520.709,E2 -15520.709} C_VEL
LIN {X 0,Y 312.455,Z 73.566,A -85,B 0,C 180,E1 -15524.209,E2 -15524.209} C_VEL
LIN {X 0,Y 312.485,Z 73.562,A -85,B 0,C 180,E1 -15527.919,E2 -15527.919} C_VEL
LIN {X 0,Y 312.497,Z 73.557,A -85,B 0,C 180,E1 -15530.97,E2 -15530.97} C_VEL
LIN {X 0,Y 312.534,Z 73.556,A -85,B 0,C 180,E1 -15534.22,E2 -15534.22} C_VEL
LIN {X 0,Y 312.55,Z 73.659,A -85,B 0,C 180,E1 -15537.896,E2 -15537.896} C_VEL
LIN {X 0,Y 315.243,Z 86.11,A -85,B 0,C 180,E1 -15541.359,E2 -15541.359} C_VEL
LIN {X 0,Y 316.46,Z 93.019,A -85,B 0,C 180,E1 -15543.203,E2 -15543.203} C_VEL
LIN {X 0,Y 315.258,Z 104.501,A -85,B 0,C 180,E1 -15546.019,E2 -15546.019} C_VEL
LIN {X 0,Y 319.631,Z 138.662,A -85,B 0,C 180,E1 -15547.125,E2 -15547.125} C_VEL
LIN {X 0,Y 320.792,Z 150.374,A -85,B 0,C 180,E1 -15547.469,E2 -15547.469} C_VEL
LIN {X 0,Y 319.573,Z 213.469,A -85,B 0,C 180,E1 -15548.892,E2 -15548.892} C_VEL
LIN {X 0,Y 318.819,Z 226.804,A -85,B 0,C 180,E1 -15549.431,E2 -15549.431} C_VEL
LIN {X 0,Y 317.851,Z 239.606,A -85,B 0,C 180,E1 -15550.21,E2 -15550.21} C_VEL
LIN {X 0,Y 316.617,Z 251.75,A -85,B 0,C 180,E1 -15551.224,E2 -15551.224} C_VEL
LIN {X 0,Y 315.311,Z 263.336,A -85,B 0,C 180,E1 -15552.488,E2 -15552.488} C_VEL
LIN {X 0,Y 314.227,Z 273.803,A -85,B 0,C 180,E1 -15553.932,E2 -15553.932} C_VEL
LIN {X 0,Y 313.319,Z 282.446,A -85,B 0,C 180,E1 -15555.404,E2 -15555.404} C_VEL
LIN {X 0,Y 312.441,Z 290.2,A -85,B 0,C 180,E1 -15557.001,E2 -15557.001} C_VEL
LIN {X 0,Y 311.558,Z 297.866,A -85,B 0,C 180,E1 -15558.945,E2 -15558.945} C_VEL
LIN {X 0,Y 311.137,Z 304.042,A -85,B 0,C 180,E1 -15560.902,E2 -15560.902} C_VEL
LIN {X 0,Y 310.836,Z 308.919,A -85,B 0,C 180,E1 -15562.856,E2 -15562.856} C_VEL
LIN {X 0,Y 310.803,Z 312.657,A -85,B 0,C 180,E1 -15564.81,E2 -15564.81} C_VEL
LIN {X 0,Y 310.864,Z 314.583,A -85,B 0,C 180,E1 -15566.111,E2 -15566.111} C_VEL
LIN {X 0,Y 310.855,Z 316.049,A -85,B 0,C 180,E1 -15567.408,E2 -15567.408} C_VEL
LIN {X 0,Y 310.948,Z 317.079,A -85,B 0,C 180,E1 -15568.705,E2 -15568.705} C_VEL
LIN {X 0,Y 311.024,Z 317.712,A -85,B 0,C 180,E1 -15570,E2 -15570} C_VEL
LIN {X 0,Y 310.871,Z 317.94,A -85,B 0,C 180,E1 -15571.295,E2 -15571.295} C_VEL
LIN {X 0,Y 310.785,Z 317.758,A -85,B 0,C 180,E1 -15572.592,E2 -15572.592} C_VEL
LIN {X 0,Y 310.782,Z 317.158,A -85,B 0,C 180,E1 -15573.89,E2 -15573.89} C_VEL
LIN {X 0,Y 310.81,Z 314.784,A -85,B 0,C 180,E1 -15576.492,E2 -15576.492} C_VEL
LIN {X 0,Y 311.084,Z 311.89,A -85,B 0,C 180,E1 -15578.444,E2 -15578.444} C_VEL
LIN {X 0,Y 311.554,Z 307.984,A -85,B 0,C 180,E1 -15580.397,E2 -15580.397} C_VEL
LIN {X 0,Y 312.352,Z 302.973,A -85,B 0,C 180,E1 -15582.342,E2 -15582.342} C_VEL
LIN {X 0,Y 313.676,Z 296.711,A -85,B 0,C 180,E1 -15584.268,E2 -15584.268} C_VEL
LIN {X 0,Y 314.995,Z 289.652,A -85,B 0,C 180,E1 -15586.027,E2 -15586.027} C_VEL
LIN {X 0,Y 316.592,Z 280.998,A -85,B 0,C 180,E1 -15587.772,E2 -15587.772} C_VEL
LIN {X 0,Y 318.445,Z 271.359,A -85,B 0,C 180,E1 -15589.332,E2 -15589.332} C_VEL
LIN {X 0,Y 320.368,Z 260.683,A -85,B 0,C 180,E1 -15590.716,E2 -15590.716} C_VEL
LIN {X 0,Y 322.024,Z 250.371,A -85,B 0,C 180,E1 -15591.778,E2 -15591.778} C_VEL
LIN {X 0,Y 323.721,Z 238.053,A -85,B 0,C 180,E1 -15592.75,E2 -15592.75} C_VEL
LIN {X 0,Y 325.098,Z 225.124,A -85,B 0,C 180,E1 -15593.49,E2 -15593.49} C_VEL
LIN {X 0,Y 325.932,Z 212.622,A -85,B 0,C 180,E1 -15593.974,E2 -15593.974} C_VEL
LIN {X 0,Y 327.631,Z 150.744,A -85,B 0,C 180,E1 -15595.361,E2 -15595.361} C_VEL
LIN {X 0,Y 324.07,Z 128.585,A -85,B 0,C 180,E1 -15596.261,E2 -15596.261} C_VEL
LIN {X 0,Y 318.955,Z 103.614,A -85,B 0,C 180,E1 -15597.443,E2 -15597.443} C_VEL
LIN {X 0,Y 318.925,Z 100.885,A -85,B 0,C 180,E1 -15598.18,E2 -15598.18} C_VEL
LIN {X 0,Y 316.607,Z 89.896,A -85,B 0,C 180,E1 -15601.443,E2 -15601.443} C_VEL
LIN {X 0,Y 314.035,Z 79.327,A -85,B 0,C 180,E1 -15604.797,E2 -15604.797} C_VEL
LIN {X 0,Y 312.525,Z 73.555,A -85,B 0,C 180,E1 -15606.76,E2 -15606.76} C_VEL
LIN {X 0,Y 312.492,Z 73.555,A -85,B 0,C 180,E1 -15610.709,E2 -15610.709} C_VEL
LIN {X 0,Y 312.454,Z 73.558,A -85,B 0,C 180,E1 -15614.21,E2 -15614.21} C_VEL
LIN {X 0,Y 312.486,Z 73.554,A -85,B 0,C 180,E1 -15617.919,E2 -15617.919} C_VEL
LIN {X 0,Y 312.508,Z 73.553,A -85,B 0,C 180,E1 -15621.917,E2 -15621.917} C_VEL
LIN {X 0,Y 312.534,Z 73.55,A -85,B 0,C 180,E1 -15624.22,E2 -15624.22} C_VEL
LIN {X 0,Y 312.507,Z 73.553,A -85,B 0,C 180,E1 -15627.334,E2 -15627.334} C_VEL
LIN {X 0,Y 312.555,Z 73.55,A -85,B 0,C 180,E1 -15631.276,E2 -15631.276} C_VEL
LIN {X 0,Y 312.589,Z 73.541,A -85,B 0,C 180,E1 -15634.711,E2 -15634.711} C_VEL
LIN {X 0,Y 312.59,Z 73.541,A -85,B 0,C 180,E1 -15637.529,E2 -15637.529} C_VEL
LIN {X 0,Y 312.641,Z 73.538,A -85,B 0,C 180,E1 -15641.656,E2 -15641.656} C_VEL
LIN {X 0,Y 312.697,Z 73.533,A -85,B 0,C 180,E1 -15645.686,E2 -15645.686} C_VEL
LIN {X 0,Y 312.702,Z 73.53,A -85,B 0,C 180,E1 -15649.642,E2 -15649.642} C_VEL
LIN {X 0,Y 312.856,Z 73.504,A -85,B 0,C 180,E1 -15652.254,E2 -15652.254} C_VEL
LIN {X 0,Y 312.715,Z 73.53,A -85,B 0,C 180,E1 -15654.842,E2 -15654.842} C_VEL
LIN {X 0,Y 312.992,Z 73.486,A -85,B 0,C 180,E1 -15658.713,E2 -15658.713} C_VEL
LIN {X 0,Y 312.992,Z 73.498,A -85,B 0,C 180,E1 -15661.286,E2 -15661.286} C_VEL
LIN {X 0,Y 312.713,Z 73.527,A -85,B 0,C 180,E1 -15665.158,E2 -15665.158} C_VEL
LIN {X 0,Y 312.884,Z 73.509,A -85,B 0,C 180,E1 -15666.548,E2 -15666.548} C_VEL
LIN {X 0,Y 312.688,Z 73.532,A -85,B 0,C 180,E1 -15670.358,E2 -15670.358} C_VEL
LIN {X 0,Y 312.67,Z 73.529,A -85,B 0,C 180,E1 -15674.865,E2 -15674.865} C_VEL
LIN {X 0,Y 312.612,Z 73.537,A -85,B 0,C 180,E1 -15679.225,E2 -15679.225} C_VEL
LIN {X 0,Y 312.547,Z 73.546,A -85,B 0,C 180,E1 -15682.789,E2 -15682.789} C_VEL
LIN {X 0,Y 312.54,Z 73.552,A -85,B 0,C 180,E1 -15685.911,E2 -15685.911} C_VEL
LIN {X 0,Y 312.505,Z 73.557,A -85,B 0,C 180,E1 -15689.654,E2 -15689.654} C_VEL
LIN {X 0,Y 312.521,Z 73.552,A -85,B 0,C 180,E1 -15693.689,E2 -15693.689} C_VEL
LIN {X 0,Y 312.516,Z 73.554,A -85,B 0,C 180,E1 -15697.386,E2 -15697.386} C_VEL
LIN {X 0,Y 312.489,Z 73.543,A -85,B 0,C 180,E1 -15700.709,E2 -15700.709} C_VEL
LIN {X 0,Y 312.452,Z 73.565,A -85,B 0,C 180,E1 -15704.209,E2 -15704.209} C_VEL
LIN {X 0,Y 312.484,Z 73.561,A -85,B 0,C 180,E1 -15707.919,E2 -15707.919} C_VEL
LIN {X 0,Y 312.492,Z 73.579,A -85,B 0,C 180,E1 -15711.368,E2 -15711.368} C_VEL
LIN {X 0,Y 312.942,Z 75.29,A -85,B 0,C 180,E1 -15711.949,E2 -15711.949} C_VEL
LIN {X 0,Y 322.273,Z 93.837,A -85,B 0,C 180,E1 -15713.463,E2 -15713.463} C_VEL
LIN {X 0,Y 328.702,Z 108.519,A -85,B 0,C 180,E1 -15714.488,E2 -15714.488} C_VEL
LIN {X 0,Y 328.135,Z 133.604,A -85,B 0,C 180,E1 -15715.052,E2 -15715.052} C_VEL
LIN {X 0,Y 326.641,Z 181.536,A -85,B 0,C 180,E1 -15716.124,E2 -15716.124} C_VEL
LIN {X 0,Y 325.886,Z 195.022,A -85,B 0,C 180,E1 -15716.684,E2 -15716.684} C_VEL
LIN {X 0,Y 325.063,Z 206.839,A -85,B 0,C 180,E1 -15717.422,E2 -15717.422} C_VEL
LIN {X 0,Y 323.786,Z 217.958,A -85,B 0,C 180,E1 -15718.325,E2 -15718.325} C_VEL
LIN {X 0,Y 322.166,Z 229.32,A -85,B 0,C 180,E1 -15719.523,E2 -15719.523} C_VEL
LIN {X 0,Y 320.447,Z 240.114,A -85,B 0,C 180,E1 -15720.972,E2 -15720.972} C_VEL
LIN {X 0,Y 318.808,Z 248.869,A -85,B 0,C 180,E1 -15722.423,E2 -15722.423} C_VEL
LIN {X 0,Y 317.26,Z 256.883,A -85,B 0,C 180,E1 -15724.055,E2 -15724.055} C_VEL
LIN {X 0,Y 315.73,Z 264.113,A -85,B 0,C 180,E1 -15725.873,E2 -15725.873} C_VEL
LIN {X 0,Y 314.425,Z 269.881,A -85,B 0,C 180,E1 -15727.667,E2 -15727.667} C_VEL
LIN {X 0,Y 313.302,Z 274.923,A -85,B 0,C 180,E1 -15729.653,E2 -15729.653} C_VEL
LIN {X 0,Y 312.461,Z 278.784,A -85,B 0,C 180,E1 -15731.646,E2 -15731.646} C_VEL
LIN {X 0,Y 311.947,Z 280.756,A -85,B 0,C 180,E1 -15732.969,E2 -15732.969} C_VEL
LIN {X 0,Y 311.566,Z 282.3,A -85,B 0,C 180,E1 -15734.295,E2 -15734.295} C_VEL
LIN {X 0,Y 311.226,Z 283.709,A -85,B 0,C 180,E1 -15736.17,E2 -15736.17} C_VEL
LIN {X 0,Y 310.91,Z 284.332,A -85,B 0,C 180,E1 -15738.262,E2 -15738.262} C_VEL
LIN {X 0,Y 310.816,Z 284.221,A -85,B 0,C 180,E1 -15739.578,E2 -15739.578} C_VEL
LIN {X 0,Y 310.839,Z 283.668,A -85,B 0,C 180,E1 -15740.894,E2 -15740.894} C_VEL
LIN {X 0,Y 311.113,Z 281.372,A -85,B 0,C 180,E1 -15743.515,E2 -15743.515} C_VEL
LIN {X 0,Y 311.246,Z 278.561,A -85,B 0,C 180,E1 -15745.467,E2 -15745.467} C_VEL
LIN {X 0,Y 311.634,Z 274.725,A -85,B 0,C 180,E1 -15747.415,E2 -15747.415} C_VEL
LIN {X 0,Y 312.037,Z 269.786,A -85,B 0,C 180,E1 -15749.355,E2 -15749.355} C_VEL
LIN {X 0,Y 312.789,Z 263.568,A -85,B 0,C 180,E1 -15751.288,E2 -15751.288} C_VEL
LIN {X 0,Y 313.728,Z 255.797,A -85,B 0,C 180,E1 -15753.211,E2 -15753.211} C_VEL
LIN {X 0,Y 314.771,Z 246.125,A -85,B 0,C 180,E1 -15755.124,E2 -15755.124} C_VEL
LIN {X 0,Y 316.034,Z 237.133,A -85,B 0,C 180,E1 -15756.544,E2 -15756.544} C_VEL
LIN {X 0,Y 317.232,Z 226.049,A -85,B 0,C 180,E1 -15757.959,E2 -15757.959} C_VEL
LIN {X 0,Y 318.229,Z 215.208,A -85,B 0,C 180,E1 -15759.053,E2 -15759.053} C_VEL
LIN {X 0,Y 319.032,Z 203.278,A -85,B 0,C 180,E1 -15759.99,E2 -15759.99} C_VEL
LIN {X 0,Y 319.629,Z 191.064,A -85,B 0,C 180,E1 -15760.692,E2 -15760.692} C_VEL
LIN {X 0,Y 320.083,Z 178.487,A -85,B 0,C 180,E1 -15761.157,E2 -15761.157} C_VEL
LIN {X 0,Y 321.586,Z 99.413,A -85,B 0,C 180,E1 -15762.923,E2 -15762.923} C_VEL
LIN {X 0,Y 313.63,Z 76.402,A -85,B 0,C 180,E1 -15763.997,E2 -15763.997} C_VEL
LIN {X 0,Y 312.757,Z 73.866,A -85,B 0,C 180,E1 -15764.126,E2 -15764.126} C_VEL
LIN {X 0,Y 312.695,Z 73.535,A -85,B 0,C 180,E1 -15764.314,E2 -15764.314} C_VEL
LIN {X 0,Y 312.639,Z 73.543,A -85,B 0,C 180,E1 -15768.344,E2 -15768.344} C_VEL
LIN {X 0,Y 312.527,Z 73.554,A -85,B 0,C 180,E1 -15772.781,E2 -15772.781} C_VEL
LIN {X 0,Y 312.604,Z 73.546,A -85,B 0,C 180,E1 -15775.936,E2 -15775.936} C_VEL
LIN {X 0,Y 312.539,Z 73.553,A -85,B 0,C 180,E1 -15779.651,E2 -15779.651} C_VEL
LIN {X 0,Y 312.521,Z 73.557,A -85,B 0,C 180,E1 -15783.689,E2 -15783.689} C_VEL
LIN {X 0,Y 312.54,Z 73.553,A -85,B 0,C 180,E1 -15787.384,E2 -15787.384} C_VEL
LIN {X 0,Y 312.492,Z 73.556,A -85,B 0,C 180,E1 -15790.709,E2 -15790.709} C_VEL
LIN {X 0,Y 312.453,Z 73.559,A -85,B 0,C 180,E1 -15793.427,E2 -15793.427} C_VEL
LIN {X 0,Y 311.778,Z 73.646,A -85,B 0,C 180,E1 -15794.504,E2 -15794.504} C_VEL
LIN {X 0,Y 308.913,Z 74.002,A -85,B 0,C 180,E1 -15796.256,E2 -15796.256} C_VEL
LIN {X 0,Y 306.509,Z 74.304,A -85,B 0,C 180,E1 -15797.676,E2 -15797.676} C_VEL
LIN {X 0,Y 305.507,Z 74.427,A -85,B 0,C 180,E1 -15798.777,E2 -15798.777} C_VEL
LIN {X 0,Y 305.442,Z 74.436,A -85,B 0,C 180,E1 -15799.149,E2 -15799.149} C_VEL
LIN {X 0,Y 305.478,Z 74.432,A -85,B 0,C 180,E1 -15801.598,E2 -15801.598} C_VEL
LIN {X 0,Y 305.465,Z 74.434,A -85,B 0,C 180,E1 -15804.887,E2 -15804.887} C_VEL
LIN {X 0,Y 305.452,Z 74.434,A -85,B 0,C 180,E1 -15808.356,E2 -15808.356} C_VEL
LIN {X 0,Y 305.516,Z 74.429,A -85,B 0,C 180,E1 -15811.114,E2 -15811.114} C_VEL
LIN {X 0,Y 305.574,Z 74.419,A -85,B 0,C 180,E1 -15814.088,E2 -15814.088} C_VEL
LIN {X 0,Y 305.505,Z 74.431,A -85,B 0,C 180,E1 -15818.403,E2 -15818.403} C_VEL
LIN {X 0,Y 305.594,Z 74.413,A -85,B 0,C 180,E1 -15821.218,E2 -15821.218} C_VEL
LIN {X 0,Y 305.653,Z 74.405,A -85,B 0,C 180,E1 -15825.349,E2 -15825.349} C_VEL
LIN {X 0,Y 305.629,Z 74.412,A -85,B 0,C 180,E1 -15829.4,E2 -15829.4} C_VEL
LIN {X 0,Y 305.791,Z 74.395,A -85,B 0,C 180,E1 -15832.074,E2 -15832.074} C_VEL
LIN {X 0,Y 305.686,Z 74.398,A -85,B 0,C 180,E1 -15834.724,E2 -15834.724} C_VEL
LIN {X 0,Y 305.959,Z 74.369,A -85,B 0,C 180,E1 -15838.684,E2 -15838.684} C_VEL
LIN {X 0,Y 305.96,Z 74.372,A -85,B 0,C 180,E1 -15841.316,E2 -15841.316} C_VEL
LIN {X 0,Y 305.675,Z 74.406,A -85,B 0,C 180,E1 -15845.277,E2 -15845.277} C_VEL
LIN {X 0,Y 305.763,Z 74.397,A -85,B 0,C 180,E1 -15847.927,E2 -15847.927} C_VEL
LIN {X 0,Y 305.603,Z 74.416,A -85,B 0,C 180,E1 -15851.945,E2 -15851.945} C_VEL
LIN {X 0,Y 305.613,Z 74.416,A -85,B 0,C 180,E1 -15855.015,E2 -15855.015} C_VEL
LIN {X 0,Y 305.564,Z 74.422,A -85,B 0,C 180,E1 -15859.436,E2 -15859.436} C_VEL
LIN {X 0,Y 305.492,Z 74.434,A -85,B 0,C 180,E1 -15863.04,E2 -15863.04} C_VEL
LIN {X 0,Y 305.481,Z 74.431,A -85,B 0,C 180,E1 -15866.2,E2 -15866.2} C_VEL
LIN {X 0,Y 305.466,Z 74.436,A -85,B 0,C 180,E1 -15869.039,E2 -15869.039} C_VEL
LIN {X 0,Y 305.44,Z 74.437,A -85,B 0,C 180,E1 -15871.953,E2 -15871.953} C_VEL
LIN {X 0,Y 305.466,Z 74.434,A -85,B 0,C 180,E1 -15875.113,E2 -15875.113} C_VEL
LIN {X 0,Y 305.453,Z 74.439,A -85,B 0,C 180,E1 -15878.529,E2 -15878.529} C_VEL
LIN {X 0,Y 305.458,Z 74.436,A -85,B 0,C 180,E1 -15882.586,E2 -15882.586} C_VEL
LIN {X 0,Y 305.428,Z 74.442,A -85,B 0,C 180,E1 -15886.345,E2 -15886.345} C_VEL
LIN {X 0,Y 305.46,Z 74.438,A -85,B 0,C 180,E1 -15889.892,E2 -15889.892} C_VEL
LIN {X 0,Y 305.481,Z 74.433,A -85,B 0,C 180,E1 -15893.632,E2 -15893.632} C_VEL
LIN {X 0,Y 305.511,Z 74.495,A -85,B 0,C 180,E1 -15897.52,E2 -15897.52} C_VEL
LIN {X 0,Y 308.187,Z 86.932,A -85,B 0,C 180,E1 -15901.07,E2 -15901.07} C_VEL
LIN {X 0,Y 309.464,Z 93.924,A -85,B 0,C 180,E1 -15902.986,E2 -15902.986} C_VEL
LIN {X 0,Y 308.409,Z 104.208,A -85,B 0,C 180,E1 -15905.571,E2 -15905.571} C_VEL
LIN {X 0,Y 313.164,Z 141.602,A -85,B 0,C 180,E1 -15906.791,E2 -15906.791} C_VEL
LIN {X 0,Y 314.059,Z 151.445,A -85,B 0,C 180,E1 -15907.082,E2 -15907.082} C_VEL
LIN {X 0,Y 312.814,Z 213.059,A -85,B 0,C 180,E1 -15908.5,E2 -15908.5} C_VEL
LIN {X 0,Y 312.045,Z 226.406,A -85,B 0,C 180,E1 -15909.05,E2 -15909.05} C_VEL
LIN {X 0,Y 311.058,Z 239.214,A -85,B 0,C 180,E1 -15909.845,E2 -15909.845} C_VEL
LIN {X 0,Y 309.891,Z 250.565,A -85,B 0,C 180,E1 -15910.801,E2 -15910.801} C_VEL
LIN {X 0,Y 308.492,Z 262.291,A -85,B 0,C 180,E1 -15912.088,E2 -15912.088} C_VEL
LIN {X 0,Y 307.331,Z 272.866,A -85,B 0,C 180,E1 -15913.561,E2 -15913.561} C_VEL
LIN {X 0,Y 306.36,Z 281.842,A -85,B 0,C 180,E1 -15915.107,E2 -15915.107} C_VEL
LIN {X 0,Y 305.477,Z 289.457,A -85,B 0,C 180,E1 -15916.699,E2 -15916.699} C_VEL
LIN {X 0,Y 304.55,Z 297.196,A -85,B 0,C 180,E1 -15918.688,E2 -15918.688} C_VEL
LIN {X 0,Y 304.072,Z 303.425,A -85,B 0,C 180,E1 -15920.689,E2 -15920.689} C_VEL
LIN {X 0,Y 303.779,Z 308.354,A -85,B 0,C 180,E1 -15922.689,E2 -15922.689} C_VEL
LIN {X 0,Y 303.707,Z 312.136,A -85,B 0,C 180,E1 -15924.689,E2 -15924.689} C_VEL
LIN {X 0,Y 303.789,Z 314.087,A -85,B 0,C 180,E1 -15926.02,E2 -15926.02} C_VEL
LIN {X 0,Y 303.772,Z 315.592,A -85,B 0,C 180,E1 -15927.348,E2 -15927.348} C_VEL
LIN {X 0,Y 303.853,Z 316.644,A -85,B 0,C 180,E1 -15928.675,E2 -15928.675} C_VEL
LIN {X 0,Y 303.933,Z 317.297,A -85,B 0,C 180,E1 -15930,E2 -15930} C_VEL
LIN {X 0,Y 303.777,Z 317.544,A -85,B 0,C 180,E1 -15931.326,E2 -15931.326} C_VEL
LIN {X 0,Y 303.703,Z 317.399,A -85,B 0,C 180,E1 -15932.653,E2 -15932.653} C_VEL
LIN {X 0,Y 303.687,Z 316.822,A -85,B 0,C 180,E1 -15933.981,E2 -15933.981} C_VEL
LIN {X 0,Y 303.723,Z 314.487,A -85,B 0,C 180,E1 -15936.644,E2 -15936.644} C_VEL
LIN {X 0,Y 304.017,Z 311.636,A -85,B 0,C 180,E1 -15938.642,E2 -15938.642} C_VEL
LIN {X 0,Y 304.546,Z 307.776,A -85,B 0,C 180,E1 -15940.639,E2 -15940.639} C_VEL
LIN {X 0,Y 305.401,Z 302.813,A -85,B 0,C 180,E1 -15942.628,E2 -15942.628} C_VEL
LIN {X 0,Y 306.77,Z 296.603,A -85,B 0,C 180,E1 -15944.596,E2 -15944.596} C_VEL
LIN {X 0,Y 308.383,Z 288.5,A -85,B 0,C 180,E1 -15946.644,E2 -15946.644} C_VEL
LIN {X 0,Y 310.172,Z 279.278,A -85,B 0,C 180,E1 -15948.495,E2 -15948.495} C_VEL
